LIN {X 21.372,Y -46.394,Z -214.360,A -90.000,B 90.000,C 0.000} C_DIS
LIN {X 21.410,Y -46.395,Z -214.288,A -90.000,B 90.000,C 0.000} C_DIS
LIN {X 22.139,Y -46.405,Z -212.980,A -90.000,B 90.000,C 0.000} C_DIS
LIN {X 23.006,Y -46.442,Z -211.414,A -90.000,B 90.000,C 0.000} C_DIS
LIN {X 23.076,Y -46.443,Z -211.265,A -90.000,B 90.000,C 0.000} C_DIS
LIN {X 23.531,Y -46.448,Z -210.300,A -90.000,B 90.000,C 0.000} C_DIS
LIN {X 23.803,Y -46.447,Z -209.727,A -90.000,B 90.000,C 0.000} C_DIS
LIN {X 23.886,Y -46.448,Z -209.562,A -90.000,B 90.000,C 0.000} C_DIS
LIN {X 24.095,Y -46.453,Z -209.183,A -90.000,B 90.000,C 0.000} C_DIS
LIN {X 24.771,Y -46.497,Z -207.945,A -90.000,B 90.000,C 0.000} C_DIS
LIN {X 25.699,Y -46.521,Z -205.750,A -90.000,B 90.000,C 0.000} C_DIS
LIN {X 25.881,Y -46.530,Z -205.318,A -90.000,B 90.000,C 0.000} C_DIS
LIN {X 25.921,Y -46.533,Z -205.229,A -90.000,B 90.000,C 0.000} C_DIS
LIN {X 26.008,Y -46.539,Z -205.045,A -90.000,B 90.000,C 0.000} C_DIS
LIN {X 26.305,Y -46.563,Z -204.477,A -90.000,B 90.000,C 0.000} C_DIS
LIN {X 27.039,Y -46.567,Z -202.392,A -90.000,B 90.000,C 0.000} C_DIS
LIN {X 27.139,Y -46.575,Z -202.102,A -90.000,B 90.000,C 0.000} C_DIS
LIN {X 27.190,Y -46.580,Z -201.966,A -90.000,B 90.000,C 0.000} C_DIS
LIN {X 27.307,Y -46.591,Z -201.675,A -90.000,B 90.000,C 0.000} C_DIS
LIN {X 27.511,Y -46.604,Z -201.180,A -90.000,B 90.000,C 0.000} C_DIS
LIN {X 27.571,Y -46.605,Z -201.006,A -90.000,B 90.000,C 0.000} C_DIS
LIN {X 28.124,Y -46.633,Z -199.578,A -90.000,B 90.000,C 0.000} C_DIS
LIN {X 28.654,Y -46.698,Z -198.194,A -90.000,B 90.000,C 0.000} C_DIS
LIN {X 28.710,Y -46.701,Z -197.852,A -90.000,B 90.000,C 0.000} C_DIS
LIN {X 28.735,Y -46.703,Z -197.715,A -90.000,B 90.000,C 0.000} C_DIS
LIN {X 28.787,Y -46.703,Z -197.474,A -90.000,B 90.000,C 0.000} C_DIS
LIN {X 28.830,Y -46.702,Z -197.310,A -90.000,B 90.000,C 0.000} C_DIS
LIN {X 28.907,Y -46.704,Z -197.051,A -90.000,B 90.000,C 0.000} C_DIS
LIN {X 28.955,Y -46.705,Z -196.908,A -90.000,B 90.000,C 0.000} C_DIS
LIN {X 28.991,Y -46.707,Z -196.811,A -90.000,B 90.000,C 0.000} C_DIS
LIN {X 29.142,Y -46.723,Z -196.407,A -90.000,B 90.000,C 0.000} C_DIS
LIN {X 29.586,Y -46.772,Z -195.213,A -90.000,B 90.000,C 0.000} C_DIS
LIN {X 29.692,Y -46.777,Z -194.390,A -90.000,B 90.000,C 0.000} C_DIS
LIN {X 29.724,Y -46.775,Z -194.150,A -90.000,B 90.000,C 0.000} C_DIS
LIN {X 29.755,Y -46.774,Z -193.950,A -90.000,B 90.000,C 0.000} C_DIS
LIN {X 29.791,Y -46.774,Z -193.778,A -90.000,B 90.000,C 0.000} C_DIS
LIN {X 29.849,Y -46.771,Z -193.528,A -90.000,B 90.000,C 0.000} C_DIS
LIN {X 29.909,Y -46.770,Z -193.322,A -90.000,B 90.000,C 0.000} C_DIS
LIN {X 30.005,Y -46.772,Z -193.045,A -90.000,B 90.000,C 0.000} C_DIS
LIN {X 30.045,Y -46.774,Z -192.940,A -90.000,B 90.000,C 0.000} C_DIS
LIN {X 30.440,Y -46.794,Z -192.024,A -90.000,B 90.000,C 0.000} C_DIS
LIN {X 30.607,Y -46.786,Z -191.348,A -90.000,B 90.000,C 0.000} C_DIS
LIN {X 30.867,Y -46.781,Z -190.293,A -90.000,B 90.000,C 0.000} C_DIS
LIN {X 30.931,Y -46.768,Z -190.045,A -90.000,B 90.000,C 0.000} C_DIS
LIN {X 30.984,Y -46.760,Z -189.864,A -90.000,B 90.000,C 0.000} C_DIS
LIN {X 31.022,Y -46.755,Z -189.755,A -90.000,B 90.000,C 0.000} C_DIS
LIN {X 31.063,Y -46.752,Z -189.652,A -90.000,B 90.000,C 0.000} C_DIS
LIN {X 31.205,Y -46.744,Z -189.325,A -90.000,B 90.000,C 0.000} C_DIS
LIN {X 31.289,Y -46.742,Z -189.154,A -90.000,B 90.000,C 0.000} C_DIS
LIN {X 31.369,Y -46.741,Z -189.007,A -90.000,B 90.000,C 0.000} C_DIS
LIN {X 31.446,Y -46.742,Z -188.873,A -90.000,B 90.000,C 0.000} C_DIS
LIN {X 32.587,Y -46.759,Z -187.003,A -90.000,B 90.000,C 0.000} C_DIS
LIN {X 32.791,Y -46.747,Z -186.673,A -90.000,B 90.000,C 0.000} C_DIS
LIN {X 33.316,Y -46.732,Z -185.855,A -90.000,B 90.000,C 0.000} C_DIS
LIN {X 33.401,Y -46.731,Z -185.733,A -90.000,B 90.000,C 0.000} C_DIS
LIN {X 33.661,Y -46.733,Z -185.402,A -90.000,B 90.000,C 0.000} C_DIS
LIN {X 33.785,Y -46.734,Z -185.258,A -90.000,B 90.000,C 0.000} C_DIS
LIN {X 34.471,Y -46.751,Z -184.535,A -90.000,B 90.000,C 0.000} C_DIS
LIN {X 34.825,Y -46.750,Z -184.164,A -90.000,B 90.000,C 0.000} C_DIS
LIN {X 35.732,Y -46.716,Z -183.029,A -90.000,B 90.000,C 0.000} C_DIS
LIN {X 35.800,Y -46.714,Z -182.948,A -90.000,B 90.000,C 0.000} C_DIS
LIN {X 35.940,Y -46.711,Z -182.790,A -90.000,B 90.000,C 0.000} C_DIS
LIN {X 36.016,Y -46.709,Z -182.708,A -90.000,B 90.000,C 0.000} C_DIS
LIN {X 36.178,Y -46.712,Z -182.543,A -90.000,B 90.000,C 0.000} C_DIS
LIN {X 36.250,Y -46.714,Z -182.474,A -90.000,B 90.000,C 0.000} C_DIS
LIN {X 36.562,Y -46.723,Z -182.187,A -90.000,B 90.000,C 0.000} C_DIS
LIN {X 37.366,Y -46.703,Z -181.213,A -90.000,B 90.000,C 0.000} C_DIS
LIN {X 37.686,Y -46.706,Z -180.823,A -90.000,B 90.000,C 0.000} C_DIS
LIN {X 37.844,Y -46.709,Z -180.642,A -90.000,B 90.000,C 0.000} C_DIS
LIN {X 38.033,Y -46.714,Z -180.443,A -90.000,B 90.000,C 0.000} C_DIS
LIN {X 38.227,Y -46.722,Z -180.255,A -90.000,B 90.000,C 0.000} C_DIS
LIN {X 38.712,Y -46.742,Z -179.794,A -90.000,B 90.000,C 0.000} C_DIS
LIN {X 39.003,Y -46.762,Z -179.516,A -90.000,B 90.000,C 0.000} C_DIS
LIN {X 39.512,Y -46.791,Z -179.030,A -90.000,B 90.000,C 0.000} C_DIS
LIN {X 39.791,Y -46.799,Z -178.695,A -90.000,B 90.000,C 0.000} C_DIS
LIN {X 39.988,Y -46.805,Z -178.453,A -90.000,B 90.000,C 0.000} C_DIS
LIN {X 40.297,Y -46.807,Z -178.072,A -90.000,B 90.000,C 0.000} C_DIS
LIN {X 40.595,Y -46.815,Z -177.702,A -90.000,B 90.000,C 0.000} C_DIS
LIN {X 41.390,Y -46.827,Z -176.606,A -90.000,B 90.000,C 0.000} C_DIS
LIN {X 41.724,Y -46.832,Z -176.114,A -90.000,B 90.000,C 0.000} C_DIS
LIN {X 42.806,Y -46.849,Z -174.449,A -90.000,B 90.000,C 0.000} C_DIS
LIN {X 42.874,Y -46.850,Z -174.341,A -90.000,B 90.000,C 0.000} C_DIS
LIN {X 43.370,Y -46.859,Z -173.506,A -90.000,B 90.000,C 0.000} C_DIS
LIN {X 44.139,Y -46.868,Z -172.255,A -90.000,B 90.000,C 0.000} C_DIS
LIN {X 44.460,Y -46.875,Z -171.698,A -90.000,B 90.000,C 0.000} C_DIS
LIN {X 44.544,Y -46.876,Z -171.552,A -90.000,B 90.000,C 0.000} C_DIS
LIN {X 44.700,Y -46.881,Z -171.303,A -90.000,B 90.000,C 0.000} C_DIS
LIN {X 44.806,Y -46.885,Z -171.151,A -90.000,B 90.000,C 0.000} C_DIS
LIN {X 44.945,Y -46.893,Z -170.968,A -90.000,B 90.000,C 0.000} C_DIS
LIN {X 45.013,Y -46.896,Z -170.884,A -90.000,B 90.000,C 0.000} C_DIS
LIN {X 45.102,Y -46.902,Z -170.782,A -90.000,B 90.000,C 0.000} C_DIS
LIN {X 45.205,Y -46.909,Z -170.673,A -90.000,B 90.000,C 0.000} C_DIS
LIN {X 45.388,Y -46.923,Z -170.496,A -90.000,B 90.000,C 0.000} C_DIS
LIN {X 45.474,Y -46.930,Z -170.421,A -90.000,B 90.000,C 0.000} C_DIS
LIN {X 45.610,Y -46.942,Z -170.310,A -90.000,B 90.000,C 0.000} C_DIS
LIN {X 45.742,Y -46.955,Z -170.211,A -90.000,B 90.000,C 0.000} C_DIS
LIN {X 45.915,Y -46.972,Z -170.093,A -90.000,B 90.000,C 0.000} C_DIS
LIN {X 47.150,Y -47.044,Z -169.316,A -90.000,B 90.000,C 0.000} C_DIS
LIN {X 48.247,Y -47.104,Z -168.572,A -90.000,B 90.000,C 0.000} C_DIS
LIN {X 48.415,Y -47.114,Z -168.462,A -90.000,B 90.000,C 0.000} C_DIS
LIN {X 48.746,Y -47.121,Z -168.040,A -90.000,B 90.000,C 0.000} C_DIS
LIN {X 48.885,Y -47.126,Z -167.874,A -90.000,B 90.000,C 0.000} C_DIS
LIN {X 48.965,Y -47.129,Z -167.783,A -90.000,B 90.000,C 0.000} C_DIS
LIN {X 49.085,Y -47.134,Z -167.660,A -90.000,B 90.000,C 0.000} C_DIS
LIN {X 49.198,Y -47.140,Z -167.558,A -90.000,B 90.000,C 0.000} C_DIS
LIN {X 49.469,Y -47.154,Z -167.331,A -90.000,B 90.000,C 0.000} C_DIS
LIN {X 49.545,Y -47.158,Z -167.271,A -90.000,B 90.000,C 0.000} C_DIS
LIN {X 49.763,Y -47.167,Z -167.118,A -90.000,B 90.000,C 0.000} C_DIS
LIN {X 49.900,Y -47.173,Z -167.026,A -90.000,B 90.000,C 0.000} C_DIS
LIN {X 50.150,Y -47.184,Z -166.876,A -90.000,B 90.000,C 0.000} C_DIS
LIN {X 50.219,Y -47.186,Z -166.840,A -90.000,B 90.000,C 0.000} C_DIS
LIN {X 50.351,Y -47.187,Z -166.775,A -90.000,B 90.000,C 0.000} C_DIS
LIN {X 50.601,Y -47.189,Z -166.668,A -90.000,B 90.000,C 0.000} C_DIS
LIN {X 50.724,Y -47.190,Z -166.620,A -90.000,B 90.000,C 0.000} C_DIS
LIN {X 50.902,Y -47.192,Z -166.561,A -90.000,B 90.000,C 0.000} C_DIS
LIN {X 51.090,Y -47.195,Z -166.509,A -90.000,B 90.000,C 0.000} C_DIS
LIN {X 51.223,Y -47.197,Z -166.478,A -90.000,B 90.000,C 0.000} C_DIS
LIN {X 51.386,Y -47.202,Z -166.453,A -90.000,B 90.000,C 0.000} C_DIS
LIN {X 51.743,Y -47.213,Z -166.406,A -90.000,B 90.000,C 0.000} C_DIS
LIN {X 51.837,Y -47.216,Z -166.396,A -90.000,B 90.000,C 0.000} C_DIS
LIN {X 51.914,Y -47.218,Z -166.391,A -90.000,B 90.000,C 0.000} C_DIS
LIN {X 52.074,Y -47.224,Z -166.388,A -90.000,B 90.000,C 0.000} C_DIS
LIN {X 52.184,Y -47.228,Z -166.390,A -90.000,B 90.000,C 0.000} C_DIS
LIN {X 52.334,Y -47.233,Z -166.397,A -90.000,B 90.000,C 0.000} C_DIS
LIN {X 52.543,Y -47.241,Z -166.416,A -90.000,B 90.000,C 0.000} C_DIS
LIN {X 52.737,Y -47.248,Z -166.445,A -90.000,B 90.000,C 0.000} C_DIS
LIN {X 52.830,Y -47.251,Z -166.462,A -90.000,B 90.000,C 0.000} C_DIS
LIN {X 53.009,Y -47.258,Z -166.501,A -90.000,B 90.000,C 0.000} C_DIS
LIN {X 53.088,Y -47.261,Z -166.522,A -90.000,B 90.000,C 0.000} C_DIS
LIN {X 53.235,Y -47.264,Z -166.563,A -90.000,B 90.000,C 0.000} C_DIS
LIN {X 53.381,Y -47.262,Z -166.611,A -90.000,B 90.000,C 0.000} C_DIS
LIN {X 53.480,Y -47.257,Z -166.648,A -90.000,B 90.000,C 0.000} C_DIS
LIN {X 53.637,Y -47.250,Z -166.710,A -90.000,B 90.000,C 0.000} C_DIS
LIN {X 53.840,Y -47.240,Z -166.805,A -90.000,B 90.000,C 0.000} C_DIS
LIN {X 53.971,Y -47.234,Z -166.872,A -90.000,B 90.000,C 0.000} C_DIS
LIN {X 54.167,Y -47.224,Z -166.990,A -90.000,B 90.000,C 0.000} C_DIS
LIN {X 54.306,Y -47.219,Z -167.076,A -90.000,B 90.000,C 0.000} C_DIS
LIN {X 54.440,Y -47.213,Z -167.172,A -90.000,B 90.000,C 0.000} C_DIS
LIN {X 54.546,Y -47.209,Z -167.254,A -90.000,B 90.000,C 0.000} C_DIS
LIN {X 54.684,Y -47.203,Z -167.367,A -90.000,B 90.000,C 0.000} C_DIS
LIN {X 54.771,Y -47.199,Z -167.448,A -90.000,B 90.000,C 0.000} C_DIS
LIN {X 54.907,Y -47.194,Z -167.577,A -90.000,B 90.000,C 0.000} C_DIS
LIN {X 55.081,Y -47.186,Z -167.767,A -90.000,B 90.000,C 0.000} C_DIS
LIN {X 55.143,Y -47.183,Z -167.838,A -90.000,B 90.000,C 0.000} C_DIS
LIN {X 55.209,Y -47.180,Z -167.921,A -90.000,B 90.000,C 0.000} C_DIS
LIN {X 55.317,Y -47.175,Z -168.064,A -90.000,B 90.000,C 0.000} C_DIS
LIN {X 55.406,Y -47.171,Z -168.195,A -90.000,B 90.000,C 0.000} C_DIS
LIN {X 55.537,Y -47.165,Z -168.411,A -90.000,B 90.000,C 0.000} C_DIS
LIN {X 55.626,Y -47.160,Z -168.579,A -90.000,B 90.000,C 0.000} C_DIS
LIN {X 55.734,Y -47.155,Z -168.807,A -90.000,B 90.000,C 0.000} C_DIS
LIN {X 55.783,Y -47.149,Z -168.928,A -90.000,B 90.000,C 0.000} C_DIS
LIN {X 55.869,Y -47.136,Z -169.161,A -90.000,B 90.000,C 0.000} C_DIS
LIN {X 55.915,Y -47.130,Z -169.299,A -90.000,B 90.000,C 0.000} C_DIS
LIN {X 55.986,Y -47.119,Z -169.530,A -90.000,B 90.000,C 0.000} C_DIS
LIN {X 56.034,Y -47.109,Z -169.718,A -90.000,B 90.000,C 0.000} C_DIS
LIN {X 56.062,Y -47.102,Z -169.849,A -90.000,B 90.000,C 0.000} C_DIS
LIN {X 56.086,Y -47.093,Z -170.031,A -90.000,B 90.000,C 0.000} C_DIS
LIN {X 56.130,Y -47.074,Z -170.524,A -90.000,B 90.000,C 0.000} C_DIS
LIN {X 56.133,Y -47.064,Z -170.838,A -90.000,B 90.000,C 0.000} C_DIS
LIN {X 56.128,Y -47.063,Z -170.904,A -90.000,B 90.000,C 0.000} C_DIS
LIN {X 56.113,Y -47.059,Z -171.088,A -90.000,B 90.000,C 0.000} C_DIS
LIN {X 55.982,Y -47.036,Z -172.370,A -90.000,B 90.000,C 0.000} C_DIS
LIN {X 55.985,Y -47.029,Z -172.609,A -90.000,B 90.000,C 0.000} C_DIS
LIN {X 55.983,Y -47.020,Z -172.904,A -90.000,B 90.000,C 0.000} C_DIS
LIN {X 55.968,Y -46.990,Z -174.748,A -90.000,B 90.000,C 0.000} C_DIS
LIN {X 56.194,Y -46.944,Z -175.853,A -90.000,B 90.000,C 0.000} C_DIS
LIN {X 56.392,Y -46.920,Z -176.820,A -90.000,B 90.000,C 0.000} C_DIS
LIN {X 56.413,Y -46.917,Z -176.933,A -90.000,B 90.000,C 0.000} C_DIS
LIN {X 56.435,Y -46.914,Z -177.003,A -90.000,B 90.000,C 0.000} C_DIS
LIN {X 56.482,Y -46.909,Z -177.157,A -90.000,B 90.000,C 0.000} C_DIS
LIN {X 56.519,Y -46.904,Z -177.291,A -90.000,B 90.000,C 0.000} C_DIS
LIN {X 56.541,Y -46.902,Z -177.397,A -90.000,B 90.000,C 0.000} C_DIS
LIN {X 56.610,Y -46.893,Z -177.772,A -90.000,B 90.000,C 0.000} C_DIS
LIN {X 56.630,Y -46.890,Z -177.901,A -90.000,B 90.000,C 0.000} C_DIS
LIN {X 56.698,Y -46.865,Z -178.691,A -90.000,B 90.000,C 0.000} C_DIS
LIN {X 56.729,Y -46.861,Z -179.054,A -90.000,B 90.000,C 0.000} C_DIS
LIN {X 56.742,Y -46.858,Z -179.247,A -90.000,B 90.000,C 0.000} C_DIS
LIN {X 56.766,Y -46.850,Z -180.111,A -90.000,B 90.000,C 0.000} C_DIS
LIN {X 56.805,Y -46.843,Z -180.308,A -90.000,B 90.000,C 0.000} C_DIS
LIN {X 56.834,Y -46.838,Z -180.478,A -90.000,B 90.000,C 0.000} C_DIS
LIN {X 56.860,Y -46.833,Z -180.668,A -90.000,B 90.000,C 0.000} C_DIS
LIN {X 56.942,Y -46.816,Z -181.375,A -90.000,B 90.000,C 0.000} C_DIS
LIN {X 57.059,Y -46.811,Z -182.378,A -90.000,B 90.000,C 0.000} C_DIS
LIN {X 57.260,Y -46.789,Z -183.172,A -90.000,B 90.000,C 0.000} C_DIS
LIN {X 57.464,Y -46.761,Z -183.982,A -90.000,B 90.000,C 0.000} C_DIS
LIN {X 57.683,Y -46.740,Z -184.857,A -90.000,B 90.000,C 0.000} C_DIS
LIN {X 57.706,Y -46.738,Z -184.961,A -90.000,B 90.000,C 0.000} C_DIS
LIN {X 57.750,Y -46.735,Z -185.198,A -90.000,B 90.000,C 0.000} C_DIS
LIN {X 57.780,Y -46.730,Z -185.418,A -90.000,B 90.000,C 0.000} C_DIS
LIN {X 57.792,Y -46.728,Z -185.529,A -90.000,B 90.000,C 0.000} C_DIS
LIN {X 57.810,Y -46.725,Z -185.751,A -90.000,B 90.000,C 0.000} C_DIS
LIN {X 57.816,Y -46.724,Z -185.862,A -90.000,B 90.000,C 0.000} C_DIS
LIN {X 57.830,Y -46.723,Z -186.394,A -90.000,B 90.000,C 0.000} C_DIS
LIN {X 57.878,Y -46.697,Z -188.394,A -90.000,B 90.000,C 0.000} C_DIS
LIN {X 57.892,Y -46.688,Z -189.117,A -90.000,B 90.000,C 0.000} C_DIS
LIN {X 57.901,Y -46.676,Z -189.755,A -90.000,B 90.000,C 0.000} C_DIS
LIN {X 57.886,Y -46.667,Z -190.472,A -90.000,B 90.000,C 0.000} C_DIS
LIN {X 57.861,Y -46.650,Z -191.585,A -90.000,B 90.000,C 0.000} C_DIS
LIN {X 57.817,Y -46.643,Z -192.376,A -90.000,B 90.000,C 0.000} C_DIS
LIN {X 57.692,Y -46.603,Z -194.422,A -90.000,B 90.000,C 0.000} C_DIS
LIN {X 57.613,Y -46.589,Z -195.317,A -90.000,B 90.000,C 0.000} C_DIS
LIN {X 57.579,Y -46.587,Z -195.575,A -90.000,B 90.000,C 0.000} C_DIS
LIN {X 57.518,Y -46.584,Z -195.936,A -90.000,B 90.000,C 0.000} C_DIS
LIN {X 57.317,Y -46.558,Z -197.358,A -90.000,B 90.000,C 0.000} C_DIS
LIN {X 57.301,Y -46.557,Z -197.457,A -90.000,B 90.000,C 0.000} C_DIS
LIN {X 57.263,Y -46.555,Z -197.652,A -90.000,B 90.000,C 0.000} C_DIS
LIN {X 57.242,Y -46.555,Z -197.750,A -90.000,B 90.000,C 0.000} C_DIS
LIN {X 56.835,Y -46.557,Z -199.423,A -90.000,B 90.000,C 0.000} C_DIS
LIN {X 56.752,Y -46.556,Z -199.758,A -90.000,B 90.000,C 0.000} C_DIS
LIN {X 56.657,Y -46.556,Z -200.089,A -90.000,B 90.000,C 0.000} C_DIS
LIN {X 55.436,Y -46.517,Z -204.266,A -90.000,B 90.000,C 0.000} C_DIS
LIN {X 55.255,Y -46.511,Z -204.846,A -90.000,B 90.000,C 0.000} C_DIS
LIN {X 53.989,Y -46.479,Z -208.784,A -90.000,B 90.000,C 0.000} C_DIS
LIN {X 53.153,Y -46.455,Z -211.322,A -90.000,B 90.000,C 0.000} C_DIS
LIN {X 52.318,Y -46.436,Z -213.780,A -90.000,B 90.000,C 0.000} C_DIS
LIN {X 51.568,Y -46.421,Z -215.923,A -90.000,B 90.000,C 0.000} C_DIS
LIN {X 50.680,Y -46.391,Z -218.613,A -90.000,B 90.000,C 0.000} C_DIS
LIN {X 50.512,Y -46.383,Z -219.120,A -90.000,B 90.000,C 0.000} C_DIS
LIN {X 50.421,Y -46.380,Z -219.365,A -90.000,B 90.000,C 0.000} C_DIS
LIN {X 49.901,Y -46.375,Z -220.611,A -90.000,B 90.000,C 0.000} C_DIS
LIN {X 48.449,Y -46.347,Z -224.309,A -90.000,B 90.000,C 0.000} C_DIS
LIN {X 48.296,Y -46.336,Z -224.688,A -90.000,B 90.000,C 0.000} C_DIS
LIN {X 48.260,Y -46.334,Z -224.769,A -90.000,B 90.000,C 0.000} C_DIS
LIN {X 48.153,Y -46.332,Z -224.986,A -90.000,B 90.000,C 0.000} C_DIS
LIN {X 47.797,Y -46.334,Z -225.635,A -90.000,B 90.000,C 0.000} C_DIS
LIN {X 45.651,Y -46.342,Z -229.733,A -90.000,B 90.000,C 0.000} C_DIS
LIN {X 45.386,Y -46.325,Z -230.225,A -90.000,B 90.000,C 0.000} C_DIS
LIN {X 45.319,Y -46.322,Z -230.340,A -90.000,B 90.000,C 0.000} C_DIS
LIN {X 45.240,Y -46.320,Z -230.470,A -90.000,B 90.000,C 0.000} C_DIS
LIN {X 45.141,Y -46.319,Z -230.620,A -90.000,B 90.000,C 0.000} C_DIS
LIN {X 45.007,Y -46.319,Z -230.811,A -90.000,B 90.000,C 0.000} C_DIS
LIN {X 44.913,Y -46.321,Z -230.936,A -90.000,B 90.000,C 0.000} C_DIS
LIN {X 44.469,Y -46.335,Z -231.506,A -90.000,B 90.000,C 0.000} C_DIS
LIN {X 42.222,Y -46.392,Z -234.502,A -90.000,B 90.000,C 0.000} C_DIS
LIN {X 42.075,Y -46.396,Z -234.697,A -90.000,B 90.000,C 0.000} C_DIS
LIN {X 41.938,Y -46.393,Z -234.877,A -90.000,B 90.000,C 0.000} C_DIS
LIN {X 41.279,Y -46.363,Z -235.736,A -90.000,B 90.000,C 0.000} C_DIS
LIN {X 41.178,Y -46.359,Z -235.859,A -90.000,B 90.000,C 0.000} C_DIS
LIN {X 40.922,Y -46.359,Z -236.132,A -90.000,B 90.000,C 0.000} C_DIS
LIN {X 40.816,Y -46.361,Z -236.236,A -90.000,B 90.000,C 0.000} C_DIS
LIN {X 40.535,Y -46.369,Z -236.493,A -90.000,B 90.000,C 0.000} C_DIS
LIN {X 39.541,Y -46.410,Z -237.341,A -90.000,B 90.000,C 0.000} C_DIS
LIN {X 37.363,Y -46.508,Z -239.204,A -90.000,B 90.000,C 0.000} C_DIS
LIN {X 37.190,Y -46.515,Z -239.357,A -90.000,B 90.000,C 0.000} C_DIS
LIN {X 35.620,Y -46.514,Z -240.714,A -90.000,B 90.000,C 0.000} C_DIS
LIN {X 35.453,Y -46.516,Z -240.850,A -90.000,B 90.000,C 0.000} C_DIS
LIN {X 35.099,Y -46.524,Z -241.116,A -90.000,B 90.000,C 0.000} C_DIS
LIN {X 34.884,Y -46.532,Z -241.266,A -90.000,B 90.000,C 0.000} C_DIS
LIN {X 34.639,Y -46.540,Z -241.425,A -90.000,B 90.000,C 0.000} C_DIS
LIN {X 34.019,Y -46.542,Z -241.822,A -90.000,B 90.000,C 0.000} C_DIS
LIN {X 32.974,Y -46.548,Z -242.464,A -90.000,B 90.000,C 0.000} C_DIS
LIN {X 32.749,Y -46.551,Z -242.591,A -90.000,B 90.000,C 0.000} C_DIS
LIN {X 32.635,Y -46.554,Z -242.650,A -90.000,B 90.000,C 0.000} C_DIS
LIN {X 32.446,Y -46.559,Z -242.740,A -90.000,B 90.000,C 0.000} C_DIS
LIN {X 32.356,Y -46.562,Z -242.780,A -90.000,B 90.000,C 0.000} C_DIS
LIN {X 32.151,Y -46.569,Z -242.866,A -90.000,B 90.000,C 0.000} C_DIS
LIN {X 32.047,Y -46.574,Z -242.906,A -90.000,B 90.000,C 0.000} C_DIS
LIN {X 30.994,Y -46.623,Z -243.279,A -90.000,B 90.000,C 0.000} C_DIS
LIN {X 30.191,Y -46.651,Z -243.561,A -90.000,B 90.000,C 0.000} C_DIS
LIN {X 30.191,Y -60.000,Z -243.561,A -90.000,B 90.000,C 0.000} C_DIS
LIN {X 14.010,Y -60.000,Z -243.561,A -90.000,B 90.000,C 0.000} C_DIS
LIN {X 14.010,Y -46.891,Z -243.561,A -90.000,B 90.000,C 0.000} C_DIS
LIN {X 13.959,Y -46.892,Z -243.476,A -90.000,B 90.000,C 0.000} C_DIS
LIN {X 13.510,Y -46.904,Z -242.722,A -90.000,B 90.000,C 0.000} C_DIS
LIN {X 13.086,Y -46.925,Z -242.012,A -90.000,B 90.000,C 0.000} C_DIS
LIN {X 13.052,Y -46.925,Z -241.955,A -90.000,B 90.000,C 0.000} C_DIS
LIN {X 12.810,Y -46.904,Z -241.545,A -90.000,B 90.000,C 0.000} C_DIS
LIN {X 11.960,Y -46.805,Z -240.098,A -90.000,B 90.000,C 0.000} C_DIS
LIN {X 11.830,Y -46.789,Z -239.865,A -90.000,B 90.000,C 0.000} C_DIS
LIN {X 11.709,Y -46.775,Z -239.631,A -90.000,B 90.000,C 0.000} C_DIS
LIN {X 11.634,Y -46.765,Z -239.474,A -90.000,B 90.000,C 0.000} C_DIS
LIN {X 11.525,Y -46.751,Z -239.218,A -90.000,B 90.000,C 0.000} C_DIS
LIN {X 11.453,Y -46.742,Z -239.014,A -90.000,B 90.000,C 0.000} C_DIS
LIN {X 11.292,Y -46.719,Z -238.497,A -90.000,B 90.000,C 0.000} C_DIS
LIN {X 11.251,Y -46.712,Z -238.354,A -90.000,B 90.000,C 0.000} C_DIS
LIN {X 11.212,Y -46.706,Z -238.196,A -90.000,B 90.000,C 0.000} C_DIS
LIN {X 11.178,Y -46.700,Z -238.026,A -90.000,B 90.000,C 0.000} C_DIS
LIN {X 11.155,Y -46.696,Z -237.892,A -90.000,B 90.000,C 0.000} C_DIS
LIN {X 11.094,Y -46.683,Z -237.451,A -90.000,B 90.000,C 0.000} C_DIS
LIN {X 11.069,Y -46.663,Z -237.257,A -90.000,B 90.000,C 0.000} C_DIS
LIN {X 11.043,Y -46.634,Z -236.968,A -90.000,B 90.000,C 0.000} C_DIS
LIN {X 11.032,Y -46.619,Z -236.802,A -90.000,B 90.000,C 0.000} C_DIS
LIN {X 11.022,Y -46.594,Z -236.521,A -90.000,B 90.000,C 0.000} C_DIS
LIN {X 11.021,Y -46.584,Z -236.407,A -90.000,B 90.000,C 0.000} C_DIS
LIN {X 11.023,Y -46.567,Z -236.192,A -90.000,B 90.000,C 0.000} C_DIS
LIN {X 11.031,Y -46.551,Z -235.982,A -90.000,B 90.000,C 0.000} C_DIS
LIN {X 11.050,Y -46.535,Z -235.754,A -90.000,B 90.000,C 0.000} C_DIS
LIN {X 11.080,Y -46.520,Z -235.513,A -90.000,B 90.000,C 0.000} C_DIS
LIN {X 11.121,Y -46.507,Z -235.265,A -90.000,B 90.000,C 0.000} C_DIS
LIN {X 11.275,Y -46.470,Z -234.509,A -90.000,B 90.000,C 0.000} C_DIS
LIN {X 12.144,Y -46.244,Z -230.270,A -90.000,B 90.000,C 0.000} C_DIS
LIN {X 12.227,Y -46.227,Z -229.912,A -90.000,B 90.000,C 0.000} C_DIS
LIN {X 12.250,Y -46.223,Z -229.820,A -90.000,B 90.000,C 0.000} C_DIS
LIN {X 12.317,Y -46.213,Z -229.582,A -90.000,B 90.000,C 0.000} C_DIS
LIN {X 12.403,Y -46.202,Z -229.309,A -90.000,B 90.000,C 0.000} C_DIS
LIN {X 12.816,Y -46.127,Z -228.037,A -90.000,B 90.000,C 0.000} C_DIS
LIN {X 13.503,Y -46.012,Z -225.913,A -90.000,B 90.000,C 0.000} C_DIS
LIN {X 13.817,Y -45.960,Z -224.949,A -90.000,B 90.000,C 0.000} C_DIS
LIN {X 13.883,Y -45.951,Z -224.768,A -90.000,B 90.000,C 0.000} C_DIS
LIN {X 13.944,Y -45.945,Z -224.611,A -90.000,B 90.000,C 0.000} C_DIS
LIN {X 14.233,Y -45.925,Z -223.939,A -90.000,B 90.000,C 0.000} C_DIS
LIN {X 14.390,Y -45.916,Z -223.580,A -90.000,B 90.000,C 0.000} C_DIS
LIN {X 15.194,Y -45.890,Z -221.928,A -90.000,B 90.000,C 0.000} C_DIS
LIN {X 16.760,Y -45.862,Z -218.903,A -90.000,B 90.000,C 0.000} C_DIS
LIN {X 17.047,Y -45.860,Z -218.348,A -90.000,B 90.000,C 0.000} C_DIS
LIN {X 17.879,Y -45.873,Z -216.819,A -90.000,B 90.000,C 0.000} C_DIS
LIN {X 19.013,Y -45.885,Z -214.742,A -90.000,B 90.000,C 0.000} C_DIS
LIN {X 19.214,Y -45.885,Z -214.344,A -90.000,B 90.000,C 0.000} C_DIS
LIN {X 19.645,Y -45.890,Z -213.488,A -90.000,B 90.000,C 0.000} C_DIS
LIN {X 19.683,Y -45.891,Z -213.415,A -90.000,B 90.000,C 0.000} C_DIS
LIN {X 20.993,Y -45.936,Z -211.047,A -90.000,B 90.000,C 0.000} C_DIS
LIN {X 21.281,Y -45.952,Z -210.524,A -90.000,B 90.000,C 0.000} C_DIS
LIN {X 22.048,Y -45.971,Z -208.895,A -90.000,B 90.000,C 0.000} C_DIS
LIN {X 22.185,Y -45.977,Z -208.623,A -90.000,B 90.000,C 0.000} C_DIS
LIN {X 22.868,Y -46.015,Z -207.373,A -90.000,B 90.000,C 0.000} C_DIS
LIN {X 23.022,Y -46.028,Z -207.089,A -90.000,B 90.000,C 0.000} C_DIS
LIN {X 23.669,Y -46.062,Z -205.549,A -90.000,B 90.000,C 0.000} C_DIS
LIN {X 24.057,Y -46.079,Z -204.630,A -90.000,B 90.000,C 0.000} C_DIS
LIN {X 24.145,Y -46.083,Z -204.427,A -90.000,B 90.000,C 0.000} C_DIS
LIN {X 24.253,Y -46.090,Z -204.197,A -90.000,B 90.000,C 0.000} C_DIS
LIN {X 24.514,Y -46.120,Z -203.690,A -90.000,B 90.000,C 0.000} C_DIS
LIN {X 25.133,Y -46.172,Z -201.901,A -90.000,B 90.000,C 0.000} C_DIS
LIN {X 25.318,Y -46.187,Z -201.374,A -90.000,B 90.000,C 0.000} C_DIS
LIN {X 25.381,Y -46.193,Z -201.207,A -90.000,B 90.000,C 0.000} C_DIS
LIN {X 25.675,Y -46.226,Z -200.481,A -90.000,B 90.000,C 0.000} C_DIS
LIN {X 25.725,Y -46.230,Z -200.334,A -90.000,B 90.000,C 0.000} C_DIS
LIN {X 26.642,Y -46.319,Z -197.945,A -90.000,B 90.000,C 0.000} C_DIS
LIN {X 26.748,Y -46.334,Z -197.667,A -90.000,B 90.000,C 0.000} C_DIS
LIN {X 26.800,Y -46.337,Z -197.364,A -90.000,B 90.000,C 0.000} C_DIS
LIN {X 26.829,Y -46.340,Z -197.222,A -90.000,B 90.000,C 0.000} C_DIS
LIN {X 26.865,Y -46.340,Z -197.058,A -90.000,B 90.000,C 0.000} C_DIS
LIN {X 26.927,Y -46.342,Z -196.812,A -90.000,B 90.000,C 0.000} C_DIS
LIN {X 27.020,Y -46.346,Z -196.493,A -90.000,B 90.000,C 0.000} C_DIS
LIN {X 27.091,Y -46.351,Z -196.276,A -90.000,B 90.000,C 0.000} C_DIS
LIN {X 27.484,Y -46.384,Z -195.219,A -90.000,B 90.000,C 0.000} C_DIS
LIN {X 27.666,Y -46.406,Z -194.730,A -90.000,B 90.000,C 0.000} C_DIS
LIN {X 27.775,Y -46.406,Z -193.896,A -90.000,B 90.000,C 0.000} C_DIS
LIN {X 27.813,Y -46.407,Z -193.646,A -90.000,B 90.000,C 0.000} C_DIS
LIN {X 27.837,Y -46.408,Z -193.520,A -90.000,B 90.000,C 0.000} C_DIS
LIN {X 27.865,Y -46.408,Z -193.381,A -90.000,B 90.000,C 0.000} C_DIS
LIN {X 27.932,Y -46.405,Z -193.089,A -90.000,B 90.000,C 0.000} C_DIS
LIN {X 27.966,Y -46.404,Z -192.962,A -90.000,B 90.000,C 0.000} C_DIS
LIN {X 28.043,Y -46.405,Z -192.699,A -90.000,B 90.000,C 0.000} C_DIS
LIN {X 28.123,Y -46.408,Z -192.468,A -90.000,B 90.000,C 0.000} C_DIS
LIN {X 28.177,Y -46.411,Z -192.317,A -90.000,B 90.000,C 0.000} C_DIS
LIN {X 28.241,Y -46.414,Z -192.155,A -90.000,B 90.000,C 0.000} C_DIS
LIN {X 28.569,Y -46.435,Z -191.392,A -90.000,B 90.000,C 0.000} C_DIS
LIN {X 28.971,Y -46.423,Z -189.765,A -90.000,B 90.000,C 0.000} C_DIS
LIN {X 29.039,Y -46.410,Z -189.503,A -90.000,B 90.000,C 0.000} C_DIS
LIN {X 29.118,Y -46.395,Z -189.244,A -90.000,B 90.000,C 0.000} C_DIS
LIN {X 29.172,Y -46.387,Z -189.089,A -90.000,B 90.000,C 0.000} C_DIS
LIN {X 29.236,Y -46.381,Z -188.927,A -90.000,B 90.000,C 0.000} C_DIS
LIN {X 29.400,Y -46.369,Z -188.549,A -90.000,B 90.000,C 0.000} C_DIS
LIN {X 29.451,Y -46.367,Z -188.442,A -90.000,B 90.000,C 0.000} C_DIS
LIN {X 29.525,Y -46.364,Z -188.291,A -90.000,B 90.000,C 0.000} C_DIS
LIN {X 29.643,Y -46.362,Z -188.071,A -90.000,B 90.000,C 0.000} C_DIS
LIN {X 29.741,Y -46.362,Z -187.899,A -90.000,B 90.000,C 0.000} C_DIS
LIN {X 30.341,Y -46.372,Z -186.913,A -90.000,B 90.000,C 0.000} C_DIS
LIN {X 30.578,Y -46.375,Z -186.525,A -90.000,B 90.000,C 0.000} C_DIS
LIN {X 31.119,Y -46.343,Z -185.653,A -90.000,B 90.000,C 0.000} C_DIS
LIN {X 31.667,Y -46.315,Z -184.804,A -90.000,B 90.000,C 0.000} C_DIS
LIN {X 31.795,Y -46.310,Z -184.619,A -90.000,B 90.000,C 0.000} C_DIS
LIN {X 31.863,Y -46.308,Z -184.528,A -90.000,B 90.000,C 0.000} C_DIS
LIN {X 32.123,Y -46.305,Z -184.197,A -90.000,B 90.000,C 0.000} C_DIS
LIN {X 32.253,Y -46.307,Z -184.041,A -90.000,B 90.000,C 0.000} C_DIS
LIN {X 32.372,Y -46.311,Z -183.907,A -90.000,B 90.000,C 0.000} C_DIS
LIN {X 32.528,Y -46.313,Z -183.743,A -90.000,B 90.000,C 0.000} C_DIS
LIN {X 33.351,Y -46.309,Z -182.883,A -90.000,B 90.000,C 0.000} C_DIS
LIN {X 33.735,Y -46.294,Z -182.402,A -90.000,B 90.000,C 0.000} C_DIS
LIN {X 34.117,Y -46.290,Z -181.920,A -90.000,B 90.000,C 0.000} C_DIS
LIN {X 34.265,Y -46.289,Z -181.736,A -90.000,B 90.000,C 0.000} C_DIS
LIN {X 34.430,Y -46.291,Z -181.546,A -90.000,B 90.000,C 0.000} C_DIS
LIN {X 34.580,Y -46.292,Z -181.380,A -90.000,B 90.000,C 0.000} C_DIS
LIN {X 34.788,Y -46.293,Z -181.168,A -90.000,B 90.000,C 0.000} C_DIS
LIN {X 34.895,Y -46.294,Z -181.064,A -90.000,B 90.000,C 0.000} C_DIS
LIN {X 35.140,Y -46.300,Z -180.838,A -90.000,B 90.000,C 0.000} C_DIS
LIN {X 36.172,Y -46.306,Z -179.579,A -90.000,B 90.000,C 0.000} C_DIS
LIN {X 36.414,Y -46.311,Z -179.302,A -90.000,B 90.000,C 0.000} C_DIS
LIN {X 36.617,Y -46.323,Z -179.087,A -90.000,B 90.000,C 0.000} C_DIS
LIN {X 36.866,Y -46.333,Z -178.842,A -90.000,B 90.000,C 0.000} C_DIS
LIN {X 37.868,Y -46.376,Z -177.890,A -90.000,B 90.000,C 0.000} C_DIS
LIN {X 38.086,Y -46.391,Z -177.682,A -90.000,B 90.000,C 0.000} C_DIS
LIN {X 38.384,Y -46.402,Z -177.320,A -90.000,B 90.000,C 0.000} C_DIS
LIN {X 39.039,Y -46.425,Z -176.506,A -90.000,B 90.000,C 0.000} C_DIS
LIN {X 39.214,Y -46.429,Z -176.265,A -90.000,B 90.000,C 0.000} C_DIS
LIN {X 39.799,Y -46.453,Z -175.453,A -90.000,B 90.000,C 0.000} C_DIS
LIN {X 40.077,Y -46.461,Z -175.041,A -90.000,B 90.000,C 0.000} C_DIS
LIN {X 40.413,Y -46.468,Z -174.525,A -90.000,B 90.000,C 0.000} C_DIS
LIN {X 41.196,Y -46.498,Z -173.312,A -90.000,B 90.000,C 0.000} C_DIS
LIN {X 41.678,Y -46.507,Z -172.498,A -90.000,B 90.000,C 0.000} C_DIS
LIN {X 42.427,Y -46.535,Z -171.273,A -90.000,B 90.000,C 0.000} C_DIS
LIN {X 42.837,Y -46.539,Z -170.565,A -90.000,B 90.000,C 0.000} C_DIS
LIN {X 43.040,Y -46.543,Z -170.240,A -90.000,B 90.000,C 0.000} C_DIS
LIN {X 43.189,Y -46.547,Z -170.022,A -90.000,B 90.000,C 0.000} C_DIS
LIN {X 43.327,Y -46.553,Z -169.838,A -90.000,B 90.000,C 0.000} C_DIS
LIN {X 43.490,Y -46.560,Z -169.632,A -90.000,B 90.000,C 0.000} C_DIS
LIN {X 43.629,Y -46.568,Z -169.471,A -90.000,B 90.000,C 0.000} C_DIS
LIN {X 43.784,Y -46.578,Z -169.305,A -90.000,B 90.000,C 0.000} C_DIS
LIN {X 43.997,Y -46.593,Z -169.097,A -90.000,B 90.000,C 0.000} C_DIS
LIN {X 44.116,Y -46.602,Z -168.986,A -90.000,B 90.000,C 0.000} C_DIS
LIN {X 44.203,Y -46.609,Z -168.911,A -90.000,B 90.000,C 0.000} C_DIS
LIN {X 44.377,Y -46.625,Z -168.767,A -90.000,B 90.000,C 0.000} C_DIS
LIN {X 44.508,Y -46.637,Z -168.667,A -90.000,B 90.000,C 0.000} C_DIS
LIN {X 44.648,Y -46.650,Z -168.565,A -90.000,B 90.000,C 0.000} C_DIS
LIN {X 44.821,Y -46.667,Z -168.447,A -90.000,B 90.000,C 0.000} C_DIS
LIN {X 46.074,Y -46.798,Z -167.648,A -90.000,B 90.000,C 0.000} C_DIS
LIN {X 46.925,Y -46.887,Z -167.065,A -90.000,B 90.000,C 0.000} C_DIS
LIN {X 47.053,Y -46.897,Z -166.978,A -90.000,B 90.000,C 0.000} C_DIS
LIN {X 47.167,Y -46.899,Z -166.833,A -90.000,B 90.000,C 0.000} C_DIS
LIN {X 47.366,Y -46.904,Z -166.591,A -90.000,B 90.000,C 0.000} C_DIS
LIN {X 47.490,Y -46.908,Z -166.452,A -90.000,B 90.000,C 0.000} C_DIS
LIN {X 47.683,Y -46.916,Z -166.250,A -90.000,B 90.000,C 0.000} C_DIS
LIN {X 47.871,Y -46.924,Z -166.077,A -90.000,B 90.000,C 0.000} C_DIS
LIN {X 48.151,Y -46.939,Z -165.841,A -90.000,B 90.000,C 0.000} C_DIS
LIN {X 48.342,Y -46.949,Z -165.687,A -90.000,B 90.000,C 0.000} C_DIS
LIN {X 48.556,Y -46.961,Z -165.534,A -90.000,B 90.000,C 0.000} C_DIS
LIN {X 48.794,Y -46.976,Z -165.371,A -90.000,B 90.000,C 0.000} C_DIS
LIN {X 48.885,Y -46.982,Z -165.313,A -90.000,B 90.000,C 0.000} C_DIS
LIN {X 49.136,Y -46.999,Z -165.162,A -90.000,B 90.000,C 0.000} C_DIS
LIN {X 49.247,Y -47.007,Z -165.100,A -90.000,B 90.000,C 0.000} C_DIS
LIN {X 49.474,Y -47.023,Z -164.985,A -90.000,B 90.000,C 0.000} C_DIS
LIN {X 49.814,Y -47.050,Z -164.834,A -90.000,B 90.000,C 0.000} C_DIS
LIN {X 49.993,Y -47.065,Z -164.762,A -90.000,B 90.000,C 0.000} C_DIS
LIN {X 50.091,Y -47.073,Z -164.726,A -90.000,B 90.000,C 0.000} C_DIS
LIN {X 50.277,Y -47.089,Z -164.664,A -90.000,B 90.000,C 0.000} C_DIS
LIN {X 50.378,Y -47.098,Z -164.633,A -90.000,B 90.000,C 0.000} C_DIS
LIN {X 50.561,Y -47.108,Z -164.582,A -90.000,B 90.000,C 0.000} C_DIS
LIN {X 50.773,Y -47.120,Z -164.531,A -90.000,B 90.000,C 0.000} C_DIS
LIN {X 50.921,Y -47.128,Z -164.503,A -90.000,B 90.000,C 0.000} C_DIS
LIN {X 51.099,Y -47.133,Z -164.475,A -90.000,B 90.000,C 0.000} C_DIS
LIN {X 51.336,Y -47.139,Z -164.444,A -90.000,B 90.000,C 0.000} C_DIS
LIN {X 51.630,Y -47.147,Z -164.408,A -90.000,B 90.000,C 0.000} C_DIS
LIN {X 51.797,Y -47.151,Z -164.395,A -90.000,B 90.000,C 0.000} C_DIS
LIN {X 52.053,Y -47.159,Z -164.389,A -90.000,B 90.000,C 0.000} C_DIS
LIN {X 52.224,Y -47.165,Z -164.391,A -90.000,B 90.000,C 0.000} C_DIS
LIN {X 52.429,Y -47.171,Z -164.400,A -90.000,B 90.000,C 0.000} C_DIS
LIN {X 52.544,Y -47.175,Z -164.409,A -90.000,B 90.000,C 0.000} C_DIS
LIN {X 52.799,Y -47.184,Z -164.434,A -90.000,B 90.000,C 0.000} C_DIS
LIN {X 52.955,Y -47.192,Z -164.456,A -90.000,B 90.000,C 0.000} C_DIS
LIN {X 53.117,Y -47.200,Z -164.482,A -90.000,B 90.000,C 0.000} C_DIS
LIN {X 53.266,Y -47.208,Z -164.510,A -90.000,B 90.000,C 0.000} C_DIS
LIN {X 53.445,Y -47.218,Z -164.550,A -90.000,B 90.000,C 0.000} C_DIS
LIN {X 53.695,Y -47.231,Z -164.615,A -90.000,B 90.000,C 0.000} C_DIS
LIN {X 53.860,Y -47.232,Z -164.663,A -90.000,B 90.000,C 0.000} C_DIS
LIN {X 53.922,Y -47.232,Z -164.684,A -90.000,B 90.000,C 0.000} C_DIS
LIN {X 54.097,Y -47.226,Z -164.743,A -90.000,B 90.000,C 0.000} C_DIS
LIN {X 54.245,Y -47.221,Z -164.800,A -90.000,B 90.000,C 0.000} C_DIS
LIN {X 54.446,Y -47.214,Z -164.882,A -90.000,B 90.000,C 0.000} C_DIS
LIN {X 54.674,Y -47.206,Z -164.987,A -90.000,B 90.000,C 0.000} C_DIS
LIN {X 54.884,Y -47.199,Z -165.093,A -90.000,B 90.000,C 0.000} C_DIS
LIN {X 54.991,Y -47.195,Z -165.153,A -90.000,B 90.000,C 0.000} C_DIS
LIN {X 55.190,Y -47.188,Z -165.271,A -90.000,B 90.000,C 0.000} C_DIS
LIN {X 55.367,Y -47.182,Z -165.381,A -90.000,B 90.000,C 0.000} C_DIS
LIN {X 55.486,Y -47.178,Z -165.462,A -90.000,B 90.000,C 0.000} C_DIS
LIN {X 55.599,Y -47.175,Z -165.542,A -90.000,B 90.000,C 0.000} C_DIS
LIN {X 55.768,Y -47.169,Z -165.671,A -90.000,B 90.000,C 0.000} C_DIS
LIN {X 55.955,Y -47.163,Z -165.823,A -90.000,B 90.000,C 0.000} C_DIS
LIN {X 56.049,Y -47.160,Z -165.907,A -90.000,B 90.000,C 0.000} C_DIS
LIN {X 56.279,Y -47.153,Z -166.122,A -90.000,B 90.000,C 0.000} C_DIS
LIN {X 56.381,Y -47.150,Z -166.226,A -90.000,B 90.000,C 0.000} C_DIS
LIN {X 56.488,Y -47.147,Z -166.342,A -90.000,B 90.000,C 0.000} C_DIS
LIN {X 56.562,Y -47.140,Z -166.423,A -90.000,B 90.000,C 0.000} C_DIS
LIN {X 56.700,Y -47.125,Z -166.584,A -90.000,B 90.000,C 0.000} C_DIS
LIN {X 56.823,Y -47.111,Z -166.743,A -90.000,B 90.000,C 0.000} C_DIS
LIN {X 56.907,Y -47.100,Z -166.853,A -90.000,B 90.000,C 0.000} C_DIS
LIN {X 57.072,Y -47.075,Z -167.092,A -90.000,B 90.000,C 0.000} C_DIS
LIN {X 57.244,Y -47.048,Z -167.375,A -90.000,B 90.000,C 0.000} C_DIS
LIN {X 57.297,Y -47.039,Z -167.470,A -90.000,B 90.000,C 0.000} C_DIS
LIN {X 57.380,Y -47.026,Z -167.627,A -90.000,B 90.000,C 0.000} C_DIS
LIN {X 57.429,Y -47.017,Z -167.725,A -90.000,B 90.000,C 0.000} C_DIS
LIN {X 57.506,Y -47.004,Z -167.888,A -90.000,B 90.000,C 0.000} C_DIS
LIN {X 57.569,Y -46.993,Z -168.028,A -90.000,B 90.000,C 0.000} C_DIS
LIN {X 57.625,Y -46.983,Z -168.166,A -90.000,B 90.000,C 0.000} C_DIS
LIN {X 57.737,Y -46.962,Z -168.469,A -90.000,B 90.000,C 0.000} C_DIS
LIN {X 57.800,Y -46.949,Z -168.654,A -90.000,B 90.000,C 0.000} C_DIS
LIN {X 57.888,Y -46.931,Z -168.942,A -90.000,B 90.000,C 0.000} C_DIS
LIN {X 57.960,Y -46.915,Z -169.216,A -90.000,B 90.000,C 0.000} C_DIS
LIN {X 58.005,Y -46.904,Z -169.418,A -90.000,B 90.000,C 0.000} C_DIS
LIN {X 58.032,Y -46.897,Z -169.575,A -90.000,B 90.000,C 0.000} C_DIS
LIN {X 58.057,Y -46.888,Z -169.757,A -90.000,B 90.000,C 0.000} C_DIS
LIN {X 58.075,Y -46.881,Z -169.944,A -90.000,B 90.000,C 0.000} C_DIS
LIN {X 58.111,Y -46.864,Z -170.350,A -90.000,B 90.000,C 0.000} C_DIS
LIN {X 58.117,Y -46.861,Z -170.441,A -90.000,B 90.000,C 0.000} C_DIS
LIN {X 58.121,Y -46.847,Z -170.836,A -90.000,B 90.000,C 0.000} C_DIS
LIN {X 58.116,Y -46.843,Z -170.970,A -90.000,B 90.000,C 0.000} C_DIS
LIN {X 58.093,Y -46.837,Z -171.251,A -90.000,B 90.000,C 0.000} C_DIS
LIN {X 57.970,Y -46.811,Z -172.453,A -90.000,B 90.000,C 0.000} C_DIS
LIN {X 57.972,Y -46.806,Z -172.577,A -90.000,B 90.000,C 0.000} C_DIS
LIN {X 57.967,Y -46.787,Z -173.205,A -90.000,B 90.000,C 0.000} C_DIS
LIN {X 57.963,Y -46.777,Z -173.786,A -90.000,B 90.000,C 0.000} C_DIS
LIN {X 57.955,Y -46.753,Z -174.550,A -90.000,B 90.000,C 0.000} C_DIS
LIN {X 58.297,Y -46.638,Z -176.253,A -90.000,B 90.000,C 0.000} C_DIS
LIN {X 58.336,Y -46.629,Z -176.450,A -90.000,B 90.000,C 0.000} C_DIS
LIN {X 58.372,Y -46.621,Z -176.570,A -90.000,B 90.000,C 0.000} C_DIS
LIN {X 58.425,Y -46.610,Z -176.761,A -90.000,B 90.000,C 0.000} C_DIS
LIN {X 58.450,Y -46.604,Z -176.867,A -90.000,B 90.000,C 0.000} C_DIS
LIN {X 58.474,Y -46.599,Z -176.979,A -90.000,B 90.000,C 0.000} C_DIS
LIN {X 58.552,Y -46.580,Z -177.407,A -90.000,B 90.000,C 0.000} C_DIS
LIN {X 58.581,Y -46.573,Z -177.601,A -90.000,B 90.000,C 0.000} C_DIS
LIN {X 58.596,Y -46.569,Z -177.722,A -90.000,B 90.000,C 0.000} C_DIS
LIN {X 58.692,Y -46.533,Z -178.856,A -90.000,B 90.000,C 0.000} C_DIS
LIN {X 58.710,Y -46.528,Z -179.117,A -90.000,B 90.000,C 0.000} C_DIS
LIN {X 58.734,Y -46.526,Z -179.885,A -90.000,B 90.000,C 0.000} C_DIS
LIN {X 58.752,Y -46.524,Z -179.981,A -90.000,B 90.000,C 0.000} C_DIS
LIN {X 58.778,Y -46.520,Z -180.136,A -90.000,B 90.000,C 0.000} C_DIS
LIN {X 58.814,Y -46.514,Z -180.383,A -90.000,B 90.000,C 0.000} C_DIS
LIN {X 58.882,Y -46.505,Z -180.958,A -90.000,B 90.000,C 0.000} C_DIS
LIN {X 59.004,Y -46.486,Z -182.014,A -90.000,B 90.000,C 0.000} C_DIS
LIN {X 59.115,Y -46.467,Z -182.459,A -90.000,B 90.000,C 0.000} C_DIS
LIN {X 59.173,Y -46.455,Z -182.693,A -90.000,B 90.000,C 0.000} C_DIS
LIN {X 59.584,Y -46.363,Z -184.361,A -90.000,B 90.000,C 0.000} C_DIS
LIN {X 59.624,Y -46.355,Z -184.542,A -90.000,B 90.000,C 0.000} C_DIS
LIN {X 59.664,Y -46.348,Z -184.760,A -90.000,B 90.000,C 0.000} C_DIS
LIN {X 59.691,Y -46.342,Z -184.920,A -90.000,B 90.000,C 0.000} C_DIS
LIN {X 59.721,Y -46.337,Z -185.139,A -90.000,B 90.000,C 0.000} C_DIS
LIN {X 59.740,Y -46.333,Z -185.310,A -90.000,B 90.000,C 0.000} C_DIS
LIN {X 59.761,Y -46.329,Z -185.556,A -90.000,B 90.000,C 0.000} C_DIS
LIN {X 59.773,Y -46.326,Z -185.754,A -90.000,B 90.000,C 0.000} C_DIS
LIN {X 59.789,Y -46.321,Z -186.342,A -90.000,B 90.000,C 0.000} C_DIS
LIN {X 59.839,Y -46.303,Z -188.353,A -90.000,B 90.000,C 0.000} C_DIS
LIN {X 59.850,Y -46.298,Z -188.927,A -90.000,B 90.000,C 0.000} C_DIS
LIN {X 59.861,Y -46.289,Z -189.596,A -90.000,B 90.000,C 0.000} C_DIS
LIN {X 59.863,Y -46.286,Z -189.798,A -90.000,B 90.000,C 0.000} C_DIS
LIN {X 59.822,Y -46.263,Z -191.632,A -90.000,B 90.000,C 0.000} C_DIS
LIN {X 59.795,Y -46.259,Z -192.137,A -90.000,B 90.000,C 0.000} C_DIS
LIN {X 59.758,Y -46.242,Z -192.755,A -90.000,B 90.000,C 0.000} C_DIS
LIN {X 59.641,Y -46.167,Z -194.533,A -90.000,B 90.000,C 0.000} C_DIS
LIN {X 59.554,Y -46.133,Z -195.481,A -90.000,B 90.000,C 0.000} C_DIS
LIN {X 59.543,Y -46.130,Z -195.571,A -90.000,B 90.000,C 0.000} C_DIS
LIN {X 59.498,Y -46.123,Z -195.895,A -90.000,B 90.000,C 0.000} C_DIS
LIN {X 59.440,Y -46.116,Z -196.228,A -90.000,B 90.000,C 0.000} C_DIS
LIN {X 59.397,Y -46.105,Z -196.529,A -90.000,B 90.000,C 0.000} C_DIS
LIN {X 59.266,Y -46.072,Z -197.424,A -90.000,B 90.000,C 0.000} C_DIS
LIN {X 59.221,Y -46.061,Z -197.719,A -90.000,B 90.000,C 0.000} C_DIS
LIN {X 59.165,Y -46.054,Z -198.013,A -90.000,B 90.000,C 0.000} C_DIS
LIN {X 59.134,Y -46.051,Z -198.159,A -90.000,B 90.000,C 0.000} C_DIS
LIN {X 58.708,Y -46.032,Z -199.889,A -90.000,B 90.000,C 0.000} C_DIS
LIN {X 58.606,Y -46.028,Z -200.290,A -90.000,B 90.000,C 0.000} C_DIS
LIN {X 57.613,Y -45.997,Z -203.693,A -90.000,B 90.000,C 0.000} C_DIS
LIN {X 57.289,Y -45.986,Z -204.802,A -90.000,B 90.000,C 0.000} C_DIS
LIN {X 57.096,Y -45.980,Z -205.418,A -90.000,B 90.000,C 0.000} C_DIS
LIN {X 55.862,Y -45.950,Z -209.259,A -90.000,B 90.000,C 0.000} C_DIS
LIN {X 54.987,Y -45.925,Z -211.920,A -90.000,B 90.000,C 0.000} C_DIS
LIN {X 54.182,Y -45.909,Z -214.288,A -90.000,B 90.000,C 0.000} C_DIS
LIN {X 53.389,Y -45.895,Z -216.561,A -90.000,B 90.000,C 0.000} C_DIS
LIN {X 52.370,Y -45.851,Z -219.638,A -90.000,B 90.000,C 0.000} C_DIS
LIN {X 52.322,Y -45.847,Z -219.780,A -90.000,B 90.000,C 0.000} C_DIS
LIN {X 52.202,Y -45.843,Z -220.099,A -90.000,B 90.000,C 0.000} C_DIS
LIN {X 51.995,Y -45.841,Z -220.596,A -90.000,B 90.000,C 0.000} C_DIS
LIN {X 51.699,Y -45.834,Z -221.301,A -90.000,B 90.000,C 0.000} C_DIS
LIN {X 50.245,Y -45.768,Z -224.972,A -90.000,B 90.000,C 0.000} C_DIS
LIN {X 50.075,Y -45.751,Z -225.389,A -90.000,B 90.000,C 0.000} C_DIS
LIN {X 50.042,Y -45.749,Z -225.466,A -90.000,B 90.000,C 0.000} C_DIS
LIN {X 49.977,Y -45.745,Z -225.610,A -90.000,B 90.000,C 0.000} C_DIS
LIN {X 49.870,Y -45.743,Z -225.827,A -90.000,B 90.000,C 0.000} C_DIS
LIN {X 49.828,Y -45.743,Z -225.908,A -90.000,B 90.000,C 0.000} C_DIS
LIN {X 49.491,Y -45.748,Z -226.523,A -90.000,B 90.000,C 0.000} C_DIS
LIN {X 48.274,Y -45.749,Z -228.844,A -90.000,B 90.000,C 0.000} C_DIS
LIN {X 47.721,Y -45.750,Z -229.901,A -90.000,B 90.000,C 0.000} C_DIS
LIN {X 47.559,Y -45.751,Z -230.209,A -90.000,B 90.000,C 0.000} C_DIS
LIN {X 47.448,Y -45.748,Z -230.420,A -90.000,B 90.000,C 0.000} C_DIS
LIN {X 47.070,Y -45.725,Z -231.122,A -90.000,B 90.000,C 0.000} C_DIS
LIN {X 47.017,Y -45.723,Z -231.214,A -90.000,B 90.000,C 0.000} C_DIS
LIN {X 46.874,Y -45.720,Z -231.454,A -90.000,B 90.000,C 0.000} C_DIS
LIN {X 46.741,Y -45.720,Z -231.661,A -90.000,B 90.000,C 0.000} C_DIS
LIN {X 46.568,Y -45.725,Z -231.911,A -90.000,B 90.000,C 0.000} C_DIS
LIN {X 46.435,Y -45.731,Z -232.092,A -90.000,B 90.000,C 0.000} C_DIS
LIN {X 45.983,Y -45.757,Z -232.677,A -90.000,B 90.000,C 0.000} C_DIS
LIN {X 43.910,Y -45.855,Z -235.463,A -90.000,B 90.000,C 0.000} C_DIS
LIN {X 43.610,Y -45.850,Z -235.858,A -90.000,B 90.000,C 0.000} C_DIS
LIN {X 42.816,Y -45.826,Z -236.897,A -90.000,B 90.000,C 0.000} C_DIS
LIN {X 42.679,Y -45.823,Z -237.068,A -90.000,B 90.000,C 0.000} C_DIS
LIN {X 42.583,Y -45.823,Z -237.178,A -90.000,B 90.000,C 0.000} C_DIS
LIN {X 42.327,Y -45.827,Z -237.452,A -90.000,B 90.000,C 0.000} C_DIS
LIN {X 42.161,Y -45.832,Z -237.618,A -90.000,B 90.000,C 0.000} C_DIS
LIN {X 41.827,Y -45.847,Z -237.927,A -90.000,B 90.000,C 0.000} C_DIS
LIN {X 41.493,Y -45.865,Z -238.215,A -90.000,B 90.000,C 0.000} C_DIS
LIN {X 39.300,Y -45.965,Z -240.092,A -90.000,B 90.000,C 0.000} C_DIS
LIN {X 38.620,Y -45.968,Z -240.663,A -90.000,B 90.000,C 0.000} C_DIS
LIN {X 37.516,Y -45.967,Z -241.617,A -90.000,B 90.000,C 0.000} C_DIS
LIN {X 36.879,Y -45.971,Z -242.170,A -90.000,B 90.000,C 0.000} C_DIS
LIN {X 36.815,Y -45.971,Z -242.223,A -90.000,B 90.000,C 0.000} C_DIS
LIN {X 36.601,Y -45.975,Z -242.396,A -90.000,B 90.000,C 0.000} C_DIS
LIN {X 36.248,Y -45.985,Z -242.662,A -90.000,B 90.000,C 0.000} C_DIS
LIN {X 35.973,Y -45.996,Z -242.855,A -90.000,B 90.000,C 0.000} C_DIS
LIN {X 35.146,Y -46.035,Z -243.399,A -90.000,B 90.000,C 0.000} C_DIS
LIN {X 34.891,Y -46.048,Z -243.561,A -90.000,B 90.000,C 0.000} C_DIS
LIN {X 34.033,Y -46.092,Z -244.113,A -90.000,B 90.000,C 0.000} C_DIS
LIN {X 33.794,Y -46.103,Z -244.270,A -90.000,B 90.000,C 0.000} C_DIS
LIN {X 33.670,Y -46.106,Z -244.358,A -90.000,B 90.000,C 0.000} C_DIS
LIN {X 33.647,Y -46.107,Z -244.375,A -90.000,B 90.000,C 0.000} C_DIS
LIN {X 33.646,Y -46.106,Z -244.379,A -90.000,B 90.000,C 0.000} C_DIS
LIN {X 33.728,Y -46.101,Z -244.339,A -90.000,B 90.000,C 0.000} C_DIS
LIN {X 33.894,Y -46.091,Z -244.245,A -90.000,B 90.000,C 0.000} C_DIS
LIN {X 36.254,Y -45.950,Z -242.843,A -90.000,B 90.000,C 0.000} C_DIS
LIN {X 37.356,Y -45.882,Z -242.198,A -90.000,B 90.000,C 0.000} C_DIS
LIN {X 37.927,Y -45.846,Z -241.868,A -90.000,B 90.000,C 0.000} C_DIS
LIN {X 39.065,Y -45.773,Z -241.221,A -90.000,B 90.000,C 0.000} C_DIS
LIN {X 39.615,Y -45.736,Z -240.915,A -90.000,B 90.000,C 0.000} C_DIS
LIN {X 40.141,Y -45.698,Z -240.629,A -90.000,B 90.000,C 0.000} C_DIS
LIN {X 40.393,Y -45.673,Z -240.495,A -90.000,B 90.000,C 0.000} C_DIS
LIN {X 40.635,Y -45.639,Z -240.368,A -90.000,B 90.000,C 0.000} C_DIS
LIN {X 40.867,Y -45.602,Z -240.249,A -90.000,B 90.000,C 0.000} C_DIS
LIN {X 41.295,Y -45.523,Z -240.036,A -90.000,B 90.000,C 0.000} C_DIS
LIN {X 41.489,Y -45.486,Z -239.945,A -90.000,B 90.000,C 0.000} C_DIS
LIN {X 41.752,Y -45.434,Z -239.827,A -90.000,B 90.000,C 0.000} C_DIS
LIN {X 41.908,Y -45.401,Z -239.763,A -90.000,B 90.000,C 0.000} C_DIS
LIN {X 42.047,Y -45.371,Z -239.711,A -90.000,B 90.000,C 0.000} C_DIS
LIN {X 42.168,Y -45.343,Z -239.672,A -90.000,B 90.000,C 0.000} C_DIS
LIN {X 42.269,Y -45.318,Z -239.646,A -90.000,B 90.000,C 0.000} C_DIS
LIN {X 42.350,Y -45.296,Z -239.635,A -90.000,B 90.000,C 0.000} C_DIS
LIN {X 42.396,Y -45.281,Z -239.637,A -90.000,B 90.000,C 0.000} C_DIS
LIN {X 42.420,Y -45.273,Z -239.642,A -90.000,B 90.000,C 0.000} C_DIS
LIN {X 42.436,Y -45.266,Z -239.651,A -90.000,B 90.000,C 0.000} C_DIS
LIN {X 42.443,Y -45.263,Z -239.658,A -90.000,B 90.000,C 0.000} C_DIS
LIN {X 42.451,Y -45.257,Z -239.673,A -90.000,B 90.000,C 0.000} C_DIS
LIN {X 42.452,Y -45.252,Z -239.692,A -90.000,B 90.000,C 0.000} C_DIS
LIN {X 42.448,Y -45.248,Z -239.715,A -90.000,B 90.000,C 0.000} C_DIS
LIN {X 42.436,Y -45.245,Z -239.744,A -90.000,B 90.000,C 0.000} C_DIS
LIN {X 42.394,Y -45.241,Z -239.817,A -90.000,B 90.000,C 0.000} C_DIS
LIN {X 42.326,Y -45.240,Z -239.909,A -90.000,B 90.000,C 0.000} C_DIS
LIN {X 42.229,Y -45.247,Z -240.019,A -90.000,B 90.000,C 0.000} C_DIS
LIN {X 42.032,Y -45.262,Z -240.223,A -90.000,B 90.000,C 0.000} C_DIS
LIN {X 41.861,Y -45.275,Z -240.386,A -90.000,B 90.000,C 0.000} C_DIS
LIN {X 41.659,Y -45.290,Z -240.571,A -90.000,B 90.000,C 0.000} C_DIS
LIN {X 41.424,Y -45.308,Z -240.779,A -90.000,B 90.000,C 0.000} C_DIS
LIN {X 41.221,Y -45.324,Z -240.955,A -90.000,B 90.000,C 0.000} C_DIS
LIN {X 39.874,Y -45.393,Z -242.112,A -90.000,B 90.000,C 0.000} C_DIS
LIN {X 38.787,Y -45.442,Z -243.070,A -90.000,B 90.000,C 0.000} C_DIS
LIN {X 38.223,Y -45.452,Z -243.561,A -90.000,B 90.000,C 0.000} C_DIS
LIN {X 38.223,Y -60.000,Z -243.561,A -90.000,B 90.000,C 0.000} C_DIS
LIN {X 11.684,Y -60.000,Z -243.561,A -90.000,B 90.000,C 0.000} C_DIS
LIN {X 11.684,Y -46.816,Z -243.561,A -90.000,B 90.000,C 0.000} C_DIS
LIN {X 11.454,Y -46.796,Z -243.173,A -90.000,B 90.000,C 0.000} C_DIS
LIN {X 10.257,Y -46.664,Z -241.138,A -90.000,B 90.000,C 0.000} C_DIS
LIN {X 10.063,Y -46.642,Z -240.790,A -90.000,B 90.000,C 0.000} C_DIS
LIN {X 9.914,Y -46.625,Z -240.500,A -90.000,B 90.000,C 0.000} C_DIS
LIN {X 9.802,Y -46.612,Z -240.262,A -90.000,B 90.000,C 0.000} C_DIS
LIN {X 9.693,Y -46.599,Z -240.006,A -90.000,B 90.000,C 0.000} C_DIS
LIN {X 9.660,Y -46.596,Z -239.924,A -90.000,B 90.000,C 0.000} C_DIS
LIN {X 9.576,Y -46.584,Z -239.687,A -90.000,B 90.000,C 0.000} C_DIS
LIN {X 9.489,Y -46.571,Z -239.412,A -90.000,B 90.000,C 0.000} C_DIS
LIN {X 9.404,Y -46.535,Z -239.132,A -90.000,B 90.000,C 0.000} C_DIS
LIN {X 9.340,Y -46.508,Z -238.906,A -90.000,B 90.000,C 0.000} C_DIS
LIN {X 9.284,Y -46.482,Z -238.677,A -90.000,B 90.000,C 0.000} C_DIS
LIN {X 9.234,Y -46.455,Z -238.429,A -90.000,B 90.000,C 0.000} C_DIS
LIN {X 9.202,Y -46.435,Z -238.237,A -90.000,B 90.000,C 0.000} C_DIS
LIN {X 9.111,Y -46.365,Z -237.533,A -90.000,B 90.000,C 0.000} C_DIS
LIN {X 9.077,Y -46.332,Z -237.176,A -90.000,B 90.000,C 0.000} C_DIS
LIN {X 9.062,Y -46.312,Z -236.960,A -90.000,B 90.000,C 0.000} C_DIS
LIN {X 9.049,Y -46.284,Z -236.639,A -90.000,B 90.000,C 0.000} C_DIS
LIN {X 9.046,Y -46.268,Z -236.450,A -90.000,B 90.000,C 0.000} C_DIS
LIN {X 9.048,Y -46.248,Z -236.198,A -90.000,B 90.000,C 0.000} C_DIS
LIN {X 9.061,Y -46.223,Z -235.874,A -90.000,B 90.000,C 0.000} C_DIS
LIN {X 9.083,Y -46.205,Z -235.611,A -90.000,B 90.000,C 0.000} C_DIS
LIN {X 9.106,Y -46.192,Z -235.411,A -90.000,B 90.000,C 0.000} C_DIS
LIN {X 9.133,Y -46.179,Z -235.210,A -90.000,B 90.000,C 0.000} C_DIS
LIN {X 9.188,Y -46.160,Z -234.889,A -90.000,B 90.000,C 0.000} C_DIS
LIN {X 9.424,Y -46.098,Z -233.735,A -90.000,B 90.000,C 0.000} C_DIS
LIN {X 9.491,Y -46.075,Z -233.411,A -90.000,B 90.000,C 0.000} C_DIS
LIN {X 9.617,Y -46.042,Z -232.797,A -90.000,B 90.000,C 0.000} C_DIS
LIN {X 9.977,Y -45.899,Z -231.092,A -90.000,B 90.000,C 0.000} C_DIS
LIN {X 10.240,Y -45.795,Z -229.851,A -90.000,B 90.000,C 0.000} C_DIS
LIN {X 10.361,Y -45.756,Z -229.357,A -90.000,B 90.000,C 0.000} C_DIS
LIN {X 10.460,Y -45.733,Z -229.016,A -90.000,B 90.000,C 0.000} C_DIS
LIN {X 11.421,Y -45.558,Z -226.051,A -90.000,B 90.000,C 0.000} C_DIS
LIN {X 11.969,Y -45.459,Z -224.373,A -90.000,B 90.000,C 0.000} C_DIS
LIN {X 12.055,Y -45.445,Z -224.133,A -90.000,B 90.000,C 0.000} C_DIS
LIN {X 12.162,Y -45.432,Z -223.862,A -90.000,B 90.000,C 0.000} C_DIS
LIN {X 12.540,Y -45.396,Z -222.994,A -90.000,B 90.000,C 0.000} C_DIS
LIN {X 12.652,Y -45.389,Z -222.743,A -90.000,B 90.000,C 0.000} C_DIS
LIN {X 13.480,Y -45.358,Z -221.045,A -90.000,B 90.000,C 0.000} C_DIS
LIN {X 14.001,Y -45.347,Z -220.039,A -90.000,B 90.000,C 0.000} C_DIS
LIN {X 14.865,Y -45.322,Z -218.377,A -90.000,B 90.000,C 0.000} C_DIS
LIN {X 15.358,Y -45.319,Z -217.423,A -90.000,B 90.000,C 0.000} C_DIS
LIN {X 15.796,Y -45.324,Z -216.619,A -90.000,B 90.000,C 0.000} C_DIS
LIN {X 17.313,Y -45.350,Z -213.834,A -90.000,B 90.000,C 0.000} C_DIS
LIN {X 17.784,Y -45.355,Z -212.897,A -90.000,B 90.000,C 0.000} C_DIS
LIN {X 17.975,Y -45.363,Z -212.518,A -90.000,B 90.000,C 0.000} C_DIS
LIN {X 19.560,Y -45.451,Z -209.636,A -90.000,B 90.000,C 0.000} C_DIS
LIN {X 19.717,Y -45.455,Z -209.302,A -90.000,B 90.000,C 0.000} C_DIS
LIN {X 19.870,Y -45.463,Z -208.974,A -90.000,B 90.000,C 0.000} C_DIS
LIN {X 20.293,Y -45.489,Z -208.065,A -90.000,B 90.000,C 0.000} C_DIS
LIN {X 20.454,Y -45.500,Z -207.741,A -90.000,B 90.000,C 0.000} C_DIS
LIN {X 21.271,Y -45.570,Z -206.232,A -90.000,B 90.000,C 0.000} C_DIS
LIN {X 21.408,Y -45.576,Z -205.907,A -90.000,B 90.000,C 0.000} C_DIS
LIN {X 21.791,Y -45.600,Z -204.993,A -90.000,B 90.000,C 0.000} C_DIS
LIN {X 22.252,Y -45.640,Z -203.888,A -90.000,B 90.000,C 0.000} C_DIS
LIN {X 22.357,Y -45.649,Z -203.641,A -90.000,B 90.000,C 0.000} C_DIS
LIN {X 22.492,Y -45.663,Z -203.353,A -90.000,B 90.000,C 0.000} C_DIS
LIN {X 22.721,Y -45.688,Z -202.904,A -90.000,B 90.000,C 0.000} C_DIS
LIN {X 22.907,Y -45.706,Z -202.364,A -90.000,B 90.000,C 0.000} C_DIS
LIN {X 23.462,Y -45.762,Z -200.759,A -90.000,B 90.000,C 0.000} C_DIS
LIN {X 23.557,Y -45.770,Z -200.502,A -90.000,B 90.000,C 0.000} C_DIS
LIN {X 23.848,Y -45.801,Z -199.785,A -90.000,B 90.000,C 0.000} C_DIS
LIN {X 23.884,Y -45.806,Z -199.676,A -90.000,B 90.000,C 0.000} C_DIS
LIN {X 24.851,Y -45.939,Z -197.135,A -90.000,B 90.000,C 0.000} C_DIS
LIN {X 24.869,Y -45.940,Z -197.030,A -90.000,B 90.000,C 0.000} C_DIS
LIN {X 24.890,Y -45.941,Z -196.923,A -90.000,B 90.000,C 0.000} C_DIS
LIN {X 24.949,Y -45.941,Z -196.644,A -90.000,B 90.000,C 0.000} C_DIS
LIN {X 25.007,Y -45.941,Z -196.411,A -90.000,B 90.000,C 0.000} C_DIS
LIN {X 25.051,Y -45.943,Z -196.244,A -90.000,B 90.000,C 0.000} C_DIS
LIN {X 25.160,Y -45.948,Z -195.874,A -90.000,B 90.000,C 0.000} C_DIS
LIN {X 25.258,Y -45.955,Z -195.581,A -90.000,B 90.000,C 0.000} C_DIS
LIN {X 25.754,Y -46.000,Z -194.248,A -90.000,B 90.000,C 0.000} C_DIS
LIN {X 25.842,Y -45.985,Z -193.600,A -90.000,B 90.000,C 0.000} C_DIS
LIN {X 25.894,Y -45.980,Z -193.279,A -90.000,B 90.000,C 0.000} C_DIS
LIN {X 25.948,Y -45.978,Z -193.005,A -90.000,B 90.000,C 0.000} C_DIS
LIN {X 26.018,Y -45.974,Z -192.698,A -90.000,B 90.000,C 0.000} C_DIS
LIN {X 26.079,Y -45.968,Z -192.463,A -90.000,B 90.000,C 0.000} C_DIS
LIN {X 26.150,Y -45.964,Z -192.223,A -90.000,B 90.000,C 0.000} C_DIS
LIN {X 26.202,Y -45.961,Z -192.056,A -90.000,B 90.000,C 0.000} C_DIS
LIN {X 26.346,Y -45.960,Z -191.652,A -90.000,B 90.000,C 0.000} C_DIS
LIN {X 26.429,Y -45.961,Z -191.438,A -90.000,B 90.000,C 0.000} C_DIS
LIN {X 26.719,Y -45.971,Z -190.767,A -90.000,B 90.000,C 0.000} C_DIS
LIN {X 26.883,Y -45.953,Z -190.116,A -90.000,B 90.000,C 0.000} C_DIS
LIN {X 27.117,Y -45.930,Z -189.188,A -90.000,B 90.000,C 0.000} C_DIS
LIN {X 27.158,Y -45.920,Z -189.034,A -90.000,B 90.000,C 0.000} C_DIS
LIN {X 27.261,Y -45.898,Z -188.693,A -90.000,B 90.000,C 0.000} C_DIS
LIN {X 27.335,Y -45.884,Z -188.478,A -90.000,B 90.000,C 0.000} C_DIS
LIN {X 27.375,Y -45.878,Z -188.372,A -90.000,B 90.000,C 0.000} C_DIS
LIN {X 27.458,Y -45.868,Z -188.170,A -90.000,B 90.000,C 0.000} C_DIS
LIN {X 27.583,Y -45.855,Z -187.884,A -90.000,B 90.000,C 0.000} C_DIS
LIN {X 27.656,Y -45.848,Z -187.722,A -90.000,B 90.000,C 0.000} C_DIS
LIN {X 27.790,Y -45.840,Z -187.447,A -90.000,B 90.000,C 0.000} C_DIS
LIN {X 27.940,Y -45.834,Z -187.165,A -90.000,B 90.000,C 0.000} C_DIS
LIN {X 28.064,Y -45.832,Z -186.947,A -90.000,B 90.000,C 0.000} C_DIS
LIN {X 28.682,Y -45.832,Z -185.936,A -90.000,B 90.000,C 0.000} C_DIS
LIN {X 29.156,Y -45.807,Z -185.173,A -90.000,B 90.000,C 0.000} C_DIS
LIN {X 29.477,Y -45.787,Z -184.655,A -90.000,B 90.000,C 0.000} C_DIS
LIN {X 30.046,Y -45.755,Z -183.775,A -90.000,B 90.000,C 0.000} C_DIS
LIN {X 30.208,Y -45.749,Z -183.538,A -90.000,B 90.000,C 0.000} C_DIS
LIN {X 30.316,Y -45.747,Z -183.390,A -90.000,B 90.000,C 0.000} C_DIS
LIN {X 30.611,Y -45.745,Z -183.013,A -90.000,B 90.000,C 0.000} C_DIS
LIN {X 30.789,Y -45.745,Z -182.800,A -90.000,B 90.000,C 0.000} C_DIS
LIN {X 30.940,Y -45.747,Z -182.629,A -90.000,B 90.000,C 0.000} C_DIS
LIN {X 31.894,Y -45.774,Z -181.619,A -90.000,B 90.000,C 0.000} C_DIS
LIN {X 32.553,Y -45.758,Z -180.790,A -90.000,B 90.000,C 0.000} C_DIS
LIN {X 32.763,Y -45.757,Z -180.528,A -90.000,B 90.000,C 0.000} C_DIS
LIN {X 32.972,Y -45.759,Z -180.284,A -90.000,B 90.000,C 0.000} C_DIS
LIN {X 33.155,Y -45.764,Z -180.081,A -90.000,B 90.000,C 0.000} C_DIS
LIN {X 33.410,Y -45.774,Z -179.815,A -90.000,B 90.000,C 0.000} C_DIS
LIN {X 33.551,Y -45.780,Z -179.675,A -90.000,B 90.000,C 0.000} C_DIS
LIN {X 33.733,Y -45.787,Z -179.505,A -90.000,B 90.000,C 0.000} C_DIS
LIN {X 34.334,Y -45.779,Z -178.777,A -90.000,B 90.000,C 0.000} C_DIS
LIN {X 34.679,Y -45.786,Z -178.353,A -90.000,B 90.000,C 0.000} C_DIS
LIN {X 34.971,Y -45.792,Z -178.018,A -90.000,B 90.000,C 0.000} C_DIS
LIN {X 35.225,Y -45.802,Z -177.748,A -90.000,B 90.000,C 0.000} C_DIS
LIN {X 35.522,Y -45.817,Z -177.454,A -90.000,B 90.000,C 0.000} C_DIS
LIN {X 35.749,Y -45.830,Z -177.237,A -90.000,B 90.000,C 0.000} C_DIS
LIN {X 36.673,Y -45.907,Z -176.346,A -90.000,B 90.000,C 0.000} C_DIS
LIN {X 36.879,Y -45.917,Z -176.094,A -90.000,B 90.000,C 0.000} C_DIS
LIN {X 37.111,Y -45.927,Z -175.806,A -90.000,B 90.000,C 0.000} C_DIS
LIN {X 37.504,Y -45.953,Z -175.313,A -90.000,B 90.000,C 0.000} C_DIS
LIN {X 38.014,Y -45.976,Z -174.604,A -90.000,B 90.000,C 0.000} C_DIS
LIN {X 38.209,Y -45.987,Z -174.331,A -90.000,B 90.000,C 0.000} C_DIS
LIN {X 38.449,Y -45.999,Z -173.974,A -90.000,B 90.000,C 0.000} C_DIS
LIN {X 39.543,Y -46.043,Z -172.281,A -90.000,B 90.000,C 0.000} C_DIS
LIN {X 40.034,Y -46.054,Z -171.454,A -90.000,B 90.000,C 0.000} C_DIS
LIN {X 40.760,Y -46.064,Z -170.274,A -90.000,B 90.000,C 0.000} C_DIS
LIN {X 41.155,Y -46.073,Z -169.588,A -90.000,B 90.000,C 0.000} C_DIS
LIN {X 41.369,Y -46.079,Z -169.243,A -90.000,B 90.000,C 0.000} C_DIS
LIN {X 41.439,Y -46.081,Z -169.134,A -90.000,B 90.000,C 0.000} C_DIS
LIN {X 41.588,Y -46.086,Z -168.916,A -90.000,B 90.000,C 0.000} C_DIS
LIN {X 41.774,Y -46.096,Z -168.664,A -90.000,B 90.000,C 0.000} C_DIS
LIN {X 41.969,Y -46.108,Z -168.415,A -90.000,B 90.000,C 0.000} C_DIS
LIN {X 42.028,Y -46.113,Z -168.342,A -90.000,B 90.000,C 0.000} C_DIS
LIN {X 42.167,Y -46.124,Z -168.182,A -90.000,B 90.000,C 0.000} C_DIS
LIN {X 42.374,Y -46.142,Z -167.956,A -90.000,B 90.000,C 0.000} C_DIS
LIN {X 42.456,Y -46.150,Z -167.873,A -90.000,B 90.000,C 0.000} C_DIS
LIN {X 42.691,Y -46.174,Z -167.641,A -90.000,B 90.000,C 0.000} C_DIS
LIN {X 42.802,Y -46.186,Z -167.537,A -90.000,B 90.000,C 0.000} C_DIS
LIN {X 42.906,Y -46.198,Z -167.444,A -90.000,B 90.000,C 0.000} C_DIS
LIN {X 43.154,Y -46.228,Z -167.236,A -90.000,B 90.000,C 0.000} C_DIS
LIN {X 43.336,Y -46.252,Z -167.093,A -90.000,B 90.000,C 0.000} C_DIS
LIN {X 43.509,Y -46.277,Z -166.963,A -90.000,B 90.000,C 0.000} C_DIS
LIN {X 43.735,Y -46.310,Z -166.805,A -90.000,B 90.000,C 0.000} C_DIS
LIN {X 44.144,Y -46.373,Z -166.540,A -90.000,B 90.000,C 0.000} C_DIS
LIN {X 44.982,Y -46.469,Z -166.004,A -90.000,B 90.000,C 0.000} C_DIS
LIN {X 45.710,Y -46.548,Z -165.505,A -90.000,B 90.000,C 0.000} C_DIS
LIN {X 45.851,Y -46.555,Z -165.333,A -90.000,B 90.000,C 0.000} C_DIS
LIN {X 46.021,Y -46.565,Z -165.138,A -90.000,B 90.000,C 0.000} C_DIS
LIN {X 46.267,Y -46.582,Z -164.878,A -90.000,B 90.000,C 0.000} C_DIS
LIN {X 46.369,Y -46.590,Z -164.778,A -90.000,B 90.000,C 0.000} C_DIS
LIN {X 46.576,Y -46.607,Z -164.587,A -90.000,B 90.000,C 0.000} C_DIS
LIN {X 46.886,Y -46.635,Z -164.322,A -90.000,B 90.000,C 0.000} C_DIS
LIN {X 47.160,Y -46.663,Z -164.099,A -90.000,B 90.000,C 0.000} C_DIS
LIN {X 47.290,Y -46.677,Z -164.004,A -90.000,B 90.000,C 0.000} C_DIS
LIN {X 47.526,Y -46.702,Z -163.836,A -90.000,B 90.000,C 0.000} C_DIS
LIN {X 47.683,Y -46.718,Z -163.728,A -90.000,B 90.000,C 0.000} C_DIS
LIN {X 47.831,Y -46.733,Z -163.631,A -90.000,B 90.000,C 0.000} C_DIS
LIN {X 48.127,Y -46.765,Z -163.452,A -90.000,B 90.000,C 0.000} C_DIS
LIN {X 48.293,Y -46.779,Z -163.358,A -90.000,B 90.000,C 0.000} C_DIS
LIN {X 48.609,Y -46.804,Z -163.195,A -90.000,B 90.000,C 0.000} C_DIS
LIN {X 49.028,Y -46.840,Z -163.007,A -90.000,B 90.000,C 0.000} C_DIS
LIN {X 49.263,Y -46.861,Z -162.911,A -90.000,B 90.000,C 0.000} C_DIS
LIN {X 49.416,Y -46.875,Z -162.854,A -90.000,B 90.000,C 0.000} C_DIS
LIN {X 49.661,Y -46.898,Z -162.771,A -90.000,B 90.000,C 0.000} C_DIS
LIN {X 49.784,Y -46.910,Z -162.732,A -90.000,B 90.000,C 0.000} C_DIS
LIN {X 50.042,Y -46.936,Z -162.659,A -90.000,B 90.000,C 0.000} C_DIS
LIN {X 50.337,Y -46.964,Z -162.586,A -90.000,B 90.000,C 0.000} C_DIS
LIN {X 50.550,Y -46.984,Z -162.543,A -90.000,B 90.000,C 0.000} C_DIS
LIN {X 50.780,Y -47.007,Z -162.505,A -90.000,B 90.000,C 0.000} C_DIS
LIN {X 51.062,Y -47.035,Z -162.465,A -90.000,B 90.000,C 0.000} C_DIS
LIN {X 51.390,Y -47.055,Z -162.424,A -90.000,B 90.000,C 0.000} C_DIS
LIN {X 51.582,Y -47.067,Z -162.408,A -90.000,B 90.000,C 0.000} C_DIS
LIN {X 51.717,Y -47.071,Z -162.399,A -90.000,B 90.000,C 0.000} C_DIS
LIN {X 52.008,Y -47.080,Z -162.391,A -90.000,B 90.000,C 0.000} C_DIS
LIN {X 52.253,Y -47.092,Z -162.393,A -90.000,B 90.000,C 0.000} C_DIS
LIN {X 52.518,Y -47.104,Z -162.403,A -90.000,B 90.000,C 0.000} C_DIS
LIN {X 52.696,Y -47.113,Z -162.416,A -90.000,B 90.000,C 0.000} C_DIS
LIN {X 52.887,Y -47.122,Z -162.434,A -90.000,B 90.000,C 0.000} C_DIS
LIN {X 53.089,Y -47.132,Z -162.456,A -90.000,B 90.000,C 0.000} C_DIS
LIN {X 53.434,Y -47.150,Z -162.508,A -90.000,B 90.000,C 0.000} C_DIS
LIN {X 53.639,Y -47.160,Z -162.546,A -90.000,B 90.000,C 0.000} C_DIS
LIN {X 53.881,Y -47.173,Z -162.599,A -90.000,B 90.000,C 0.000} C_DIS
LIN {X 54.258,Y -47.194,Z -162.696,A -90.000,B 90.000,C 0.000} C_DIS
LIN {X 54.360,Y -47.196,Z -162.726,A -90.000,B 90.000,C 0.000} C_DIS
LIN {X 54.494,Y -47.196,Z -162.767,A -90.000,B 90.000,C 0.000} C_DIS
LIN {X 54.729,Y -47.188,Z -162.846,A -90.000,B 90.000,C 0.000} C_DIS
LIN {X 54.916,Y -47.183,Z -162.916,A -90.000,B 90.000,C 0.000} C_DIS
LIN {X 55.192,Y -47.176,Z -163.026,A -90.000,B 90.000,C 0.000} C_DIS
LIN {X 55.289,Y -47.173,Z -163.068,A -90.000,B 90.000,C 0.000} C_DIS
LIN {X 55.517,Y -47.168,Z -163.174,A -90.000,B 90.000,C 0.000} C_DIS
LIN {X 55.781,Y -47.161,Z -163.306,A -90.000,B 90.000,C 0.000} C_DIS
LIN {X 55.959,Y -47.157,Z -163.403,A -90.000,B 90.000,C 0.000} C_DIS
LIN {X 56.163,Y -47.152,Z -163.523,A -90.000,B 90.000,C 0.000} C_DIS
LIN {X 56.408,Y -47.146,Z -163.674,A -90.000,B 90.000,C 0.000} C_DIS
LIN {X 56.607,Y -47.141,Z -163.806,A -90.000,B 90.000,C 0.000} C_DIS
LIN {X 56.819,Y -47.136,Z -163.958,A -90.000,B 90.000,C 0.000} C_DIS
LIN {X 57.039,Y -47.131,Z -164.127,A -90.000,B 90.000,C 0.000} C_DIS
LIN {X 57.140,Y -47.128,Z -164.209,A -90.000,B 90.000,C 0.000} C_DIS
LIN {X 57.287,Y -47.114,Z -164.333,A -90.000,B 90.000,C 0.000} C_DIS
LIN {X 57.435,Y -47.100,Z -164.466,A -90.000,B 90.000,C 0.000} C_DIS
LIN {X 57.645,Y -47.076,Z -164.663,A -90.000,B 90.000,C 0.000} C_DIS
LIN {X 57.799,Y -47.057,Z -164.818,A -90.000,B 90.000,C 0.000} C_DIS
LIN {X 58.031,Y -47.028,Z -165.071,A -90.000,B 90.000,C 0.000} C_DIS
LIN {X 58.249,Y -47.001,Z -165.325,A -90.000,B 90.000,C 0.000} C_DIS
LIN {X 58.493,Y -46.969,Z -165.642,A -90.000,B 90.000,C 0.000} C_DIS
LIN {X 58.707,Y -46.941,Z -165.948,A -90.000,B 90.000,C 0.000} C_DIS
LIN {X 58.770,Y -46.932,Z -166.045,A -90.000,B 90.000,C 0.000} C_DIS
LIN {X 58.943,Y -46.908,Z -166.329,A -90.000,B 90.000,C 0.000} C_DIS
LIN {X 59.029,Y -46.896,Z -166.480,A -90.000,B 90.000,C 0.000} C_DIS
LIN {X 59.152,Y -46.879,Z -166.710,A -90.000,B 90.000,C 0.000} C_DIS
LIN {X 59.250,Y -46.865,Z -166.910,A -90.000,B 90.000,C 0.000} C_DIS
LIN {X 59.308,Y -46.855,Z -167.035,A -90.000,B 90.000,C 0.000} C_DIS
LIN {X 59.416,Y -46.836,Z -167.278,A -90.000,B 90.000,C 0.000} C_DIS
LIN {X 59.467,Y -46.826,Z -167.403,A -90.000,B 90.000,C 0.000} C_DIS
LIN {X 59.603,Y -46.800,Z -167.769,A -90.000,B 90.000,C 0.000} C_DIS
LIN {X 59.717,Y -46.777,Z -168.108,A -90.000,B 90.000,C 0.000} C_DIS
LIN {X 59.789,Y -46.752,Z -168.348,A -90.000,B 90.000,C 0.000} C_DIS
LIN {X 59.882,Y -46.717,Z -168.699,A -90.000,B 90.000,C 0.000} C_DIS
LIN {X 59.944,Y -46.692,Z -168.974,A -90.000,B 90.000,C 0.000} C_DIS
LIN {X 59.963,Y -46.683,Z -169.078,A -90.000,B 90.000,C 0.000} C_DIS
LIN {X 59.994,Y -46.668,Z -169.258,A -90.000,B 90.000,C 0.000} C_DIS
LIN {X 60.031,Y -46.645,Z -169.551,A -90.000,B 90.000,C 0.000} C_DIS
LIN {X 60.040,Y -46.639,Z -169.645,A -90.000,B 90.000,C 0.000} C_DIS
LIN {X 60.089,Y -46.599,Z -170.219,A -90.000,B 90.000,C 0.000} C_DIS
LIN {X 60.098,Y -46.587,Z -170.410,A -90.000,B 90.000,C 0.000} C_DIS
LIN {X 60.101,Y -46.565,Z -170.805,A -90.000,B 90.000,C 0.000} C_DIS
LIN {X 60.094,Y -46.554,Z -171.032,A -90.000,B 90.000,C 0.000} C_DIS
LIN {X 60.089,Y -46.550,Z -171.121,A -90.000,B 90.000,C 0.000} C_DIS
LIN {X 60.065,Y -46.539,Z -171.402,A -90.000,B 90.000,C 0.000} C_DIS
LIN {X 59.948,Y -46.499,Z -172.534,A -90.000,B 90.000,C 0.000} C_DIS
LIN {X 59.936,Y -46.448,Z -173.580,A -90.000,B 90.000,C 0.000} C_DIS
LIN {X 59.929,Y -46.425,Z -174.347,A -90.000,B 90.000,C 0.000} C_DIS
LIN {X 60.251,Y -46.318,Z -175.955,A -90.000,B 90.000,C 0.000} C_DIS
LIN {X 60.325,Y -46.297,Z -176.222,A -90.000,B 90.000,C 0.000} C_DIS
LIN {X 60.366,Y -46.285,Z -176.389,A -90.000,B 90.000,C 0.000} C_DIS
LIN {X 60.412,Y -46.270,Z -176.614,A -90.000,B 90.000,C 0.000} C_DIS
LIN {X 60.490,Y -46.250,Z -177.039,A -90.000,B 90.000,C 0.000} C_DIS
LIN {X 60.529,Y -46.239,Z -177.289,A -90.000,B 90.000,C 0.000} C_DIS
LIN {X 60.553,Y -46.230,Z -177.494,A -90.000,B 90.000,C 0.000} C_DIS
LIN {X 60.605,Y -46.210,Z -178.090,A -90.000,B 90.000,C 0.000} C_DIS
LIN {X 60.654,Y -46.184,Z -178.678,A -90.000,B 90.000,C 0.000} C_DIS
LIN {X 60.673,Y -46.172,Z -178.979,A -90.000,B 90.000,C 0.000} C_DIS
LIN {X 60.684,Y -46.160,Z -179.355,A -90.000,B 90.000,C 0.000} C_DIS
LIN {X 60.693,Y -46.156,Z -179.674,A -90.000,B 90.000,C 0.000} C_DIS
LIN {X 60.714,Y -46.150,Z -179.794,A -90.000,B 90.000,C 0.000} C_DIS
LIN {X 60.757,Y -46.138,Z -180.092,A -90.000,B 90.000,C 0.000} C_DIS
LIN {X 60.933,Y -46.082,Z -181.651,A -90.000,B 90.000,C 0.000} C_DIS
LIN {X 61.011,Y -46.062,Z -181.966,A -90.000,B 90.000,C 0.000} C_DIS
LIN {X 61.497,Y -45.962,Z -183.936,A -90.000,B 90.000,C 0.000} C_DIS
LIN {X 61.534,Y -45.955,Z -184.108,A -90.000,B 90.000,C 0.000} C_DIS
LIN {X 61.587,Y -45.943,Z -184.391,A -90.000,B 90.000,C 0.000} C_DIS
LIN {X 61.619,Y -45.935,Z -184.580,A -90.000,B 90.000,C 0.000} C_DIS
LIN {X 61.666,Y -45.926,Z -184.918,A -90.000,B 90.000,C 0.000} C_DIS
LIN {X 61.682,Y -45.923,Z -185.060,A -90.000,B 90.000,C 0.000} C_DIS
LIN {X 61.711,Y -45.917,Z -185.386,A -90.000,B 90.000,C 0.000} C_DIS
LIN {X 61.726,Y -45.915,Z -185.630,A -90.000,B 90.000,C 0.000} C_DIS
LIN {X 61.746,Y -45.913,Z -186.328,A -90.000,B 90.000,C 0.000} C_DIS
LIN {X 61.768,Y -45.889,Z -187.323,A -90.000,B 90.000,C 0.000} C_DIS
LIN {X 61.788,Y -45.857,Z -188.312,A -90.000,B 90.000,C 0.000} C_DIS
LIN {X 61.804,Y -45.817,Z -189.574,A -90.000,B 90.000,C 0.000} C_DIS
LIN {X 61.805,Y -45.811,Z -189.776,A -90.000,B 90.000,C 0.000} C_DIS
LIN {X 61.796,Y -45.802,Z -190.189,A -90.000,B 90.000,C 0.000} C_DIS
LIN {X 61.752,Y -45.747,Z -191.726,A -90.000,B 90.000,C 0.000} C_DIS
LIN {X 61.668,Y -45.709,Z -193.118,A -90.000,B 90.000,C 0.000} C_DIS
LIN {X 61.568,Y -45.644,Z -194.637,A -90.000,B 90.000,C 0.000} C_DIS
LIN {X 61.477,Y -45.608,Z -195.637,A -90.000,B 90.000,C 0.000} C_DIS
LIN {X 61.462,Y -45.604,Z -195.776,A -90.000,B 90.000,C 0.000} C_DIS
LIN {X 61.410,Y -45.595,Z -196.152,A -90.000,B 90.000,C 0.000} C_DIS
LIN {X 61.356,Y -45.590,Z -196.473,A -90.000,B 90.000,C 0.000} C_DIS
LIN {X 61.264,Y -45.568,Z -197.091,A -90.000,B 90.000,C 0.000} C_DIS
LIN {X 61.131,Y -45.535,Z -197.991,A -90.000,B 90.000,C 0.000} C_DIS
LIN {X 61.063,Y -45.525,Z -198.359,A -90.000,B 90.000,C 0.000} C_DIS
LIN {X 61.007,Y -45.520,Z -198.617,A -90.000,B 90.000,C 0.000} C_DIS
LIN {X 60.582,Y -45.502,Z -200.344,A -90.000,B 90.000,C 0.000} C_DIS
LIN {X 60.517,Y -45.499,Z -200.599,A -90.000,B 90.000,C 0.000} C_DIS
LIN {X 60.458,Y -45.495,Z -200.824,A -90.000,B 90.000,C 0.000} C_DIS
LIN {X 59.396,Y -45.454,Z -204.457,A -90.000,B 90.000,C 0.000} C_DIS
LIN {X 59.135,Y -45.434,Z -205.336,A -90.000,B 90.000,C 0.000} C_DIS
LIN {X 58.930,Y -45.420,Z -205.986,A -90.000,B 90.000,C 0.000} C_DIS
LIN {X 57.676,Y -45.350,Z -209.850,A -90.000,B 90.000,C 0.000} C_DIS
LIN {X 57.023,Y -45.308,Z -211.810,A -90.000,B 90.000,C 0.000} C_DIS
LIN {X 57.023,Y -60.000,Z -211.810,A -90.000,B 90.000,C 0.000} C_DIS
LIN {X 35.139,Y -60.000,Z -175.166,A -90.000,B 90.000,C 0.000} C_DIS
LIN {X 35.139,Y -45.308,Z -175.166,A -90.000,B 90.000,C 0.000} C_DIS
LIN {X 35.282,Y -45.326,Z -175.026,A -90.000,B 90.000,C 0.000} C_DIS
LIN {X 35.544,Y -45.346,Z -174.699,A -90.000,B 90.000,C 0.000} C_DIS
LIN {X 36.000,Y -45.375,Z -174.127,A -90.000,B 90.000,C 0.000} C_DIS
LIN {X 36.555,Y -45.413,Z -173.348,A -90.000,B 90.000,C 0.000} C_DIS
LIN {X 36.645,Y -45.417,Z -173.223,A -90.000,B 90.000,C 0.000} C_DIS
LIN {X 36.858,Y -45.423,Z -172.908,A -90.000,B 90.000,C 0.000} C_DIS
LIN {X 37.367,Y -45.433,Z -172.127,A -90.000,B 90.000,C 0.000} C_DIS
LIN {X 37.602,Y -45.442,Z -171.763,A -90.000,B 90.000,C 0.000} C_DIS
LIN {X 37.924,Y -45.451,Z -171.266,A -90.000,B 90.000,C 0.000} C_DIS
LIN {X 38.411,Y -45.455,Z -170.450,A -90.000,B 90.000,C 0.000} C_DIS
LIN {X 38.659,Y -45.460,Z -170.045,A -90.000,B 90.000,C 0.000} C_DIS
LIN {X 39.127,Y -45.478,Z -169.278,A -90.000,B 90.000,C 0.000} C_DIS
LIN {X 39.503,Y -45.486,Z -168.627,A -90.000,B 90.000,C 0.000} C_DIS
LIN {X 39.765,Y -45.496,Z -168.201,A -90.000,B 90.000,C 0.000} C_DIS
LIN {X 39.871,Y -45.502,Z -168.037,A -90.000,B 90.000,C 0.000} C_DIS
LIN {X 40.023,Y -45.510,Z -167.813,A -90.000,B 90.000,C 0.000} C_DIS
LIN {X 40.277,Y -45.527,Z -167.466,A -90.000,B 90.000,C 0.000} C_DIS
LIN {X 40.471,Y -45.542,Z -167.216,A -90.000,B 90.000,C 0.000} C_DIS
LIN {X 40.550,Y -45.550,Z -167.119,A -90.000,B 90.000,C 0.000} C_DIS
LIN {X 40.775,Y -45.572,Z -166.855,A -90.000,B 90.000,C 0.000} C_DIS
LIN {X 40.979,Y -45.596,Z -166.631,A -90.000,B 90.000,C 0.000} C_DIS
LIN {X 41.109,Y -45.613,Z -166.495,A -90.000,B 90.000,C 0.000} C_DIS
LIN {X 41.400,Y -45.655,Z -166.204,A -90.000,B 90.000,C 0.000} C_DIS
LIN {X 41.566,Y -45.681,Z -166.048,A -90.000,B 90.000,C 0.000} C_DIS
LIN {X 41.705,Y -45.702,Z -165.924,A -90.000,B 90.000,C 0.000} C_DIS
LIN {X 41.996,Y -45.741,Z -165.680,A -90.000,B 90.000,C 0.000} C_DIS
LIN {X 42.178,Y -45.766,Z -165.536,A -90.000,B 90.000,C 0.000} C_DIS
LIN {X 42.409,Y -45.800,Z -165.362,A -90.000,B 90.000,C 0.000} C_DIS
LIN {X 42.702,Y -45.845,Z -165.157,A -90.000,B 90.000,C 0.000} C_DIS
LIN {X 43.938,Y -46.041,Z -164.352,A -90.000,B 90.000,C 0.000} C_DIS
LIN {X 44.399,Y -46.111,Z -164.032,A -90.000,B 90.000,C 0.000} C_DIS
LIN {X 44.563,Y -46.125,Z -163.842,A -90.000,B 90.000,C 0.000} C_DIS
LIN {X 44.617,Y -46.131,Z -163.782,A -90.000,B 90.000,C 0.000} C_DIS
LIN {X 44.861,Y -46.157,Z -163.521,A -90.000,B 90.000,C 0.000} C_DIS
LIN {X 45.017,Y -46.175,Z -163.364,A -90.000,B 90.000,C 0.000} C_DIS
LIN {X 45.262,Y -46.205,Z -163.134,A -90.000,B 90.000,C 0.000} C_DIS
LIN {X 45.418,Y -46.225,Z -162.996,A -90.000,B 90.000,C 0.000} C_DIS
LIN {X 45.589,Y -46.242,Z -162.850,A -90.000,B 90.000,C 0.000} C_DIS
LIN {X 45.945,Y -46.278,Z -162.558,A -90.000,B 90.000,C 0.000} C_DIS
LIN {X 46.057,Y -46.290,Z -162.473,A -90.000,B 90.000,C 0.000} C_DIS
LIN {X 46.232,Y -46.309,Z -162.346,A -90.000,B 90.000,C 0.000} C_DIS
LIN {X 46.590,Y -46.350,Z -162.094,A -90.000,B 90.000,C 0.000} C_DIS
LIN {X 46.799,Y -46.375,Z -161.956,A -90.000,B 90.000,C 0.000} C_DIS
LIN {X 47.178,Y -46.423,Z -161.725,A -90.000,B 90.000,C 0.000} C_DIS
LIN {X 47.412,Y -46.453,Z -161.592,A -90.000,B 90.000,C 0.000} C_DIS
LIN {X 47.725,Y -46.495,Z -161.428,A -90.000,B 90.000,C 0.000} C_DIS
LIN {X 47.822,Y -46.509,Z -161.380,A -90.000,B 90.000,C 0.000} C_DIS
LIN {X 48.239,Y -46.568,Z -161.189,A -90.000,B 90.000,C 0.000} C_DIS
LIN {X 48.533,Y -46.608,Z -161.066,A -90.000,B 90.000,C 0.000} C_DIS
LIN {X 48.737,Y -46.633,Z -160.988,A -90.000,B 90.000,C 0.000} C_DIS
LIN {X 49.043,Y -46.669,Z -160.882,A -90.000,B 90.000,C 0.000} C_DIS
LIN {X 49.275,Y -46.693,Z -160.810,A -90.000,B 90.000,C 0.000} C_DIS
LIN {X 49.583,Y -46.725,Z -160.724,A -90.000,B 90.000,C 0.000} C_DIS
LIN {X 49.878,Y -46.755,Z -160.650,A -90.000,B 90.000,C 0.000} C_DIS
LIN {X 50.174,Y -46.785,Z -160.588,A -90.000,B 90.000,C 0.000} C_DIS
LIN {X 50.476,Y -46.818,Z -160.537,A -90.000,B 90.000,C 0.000} C_DIS
LIN {X 50.553,Y -46.826,Z -160.526,A -90.000,B 90.000,C 0.000} C_DIS
LIN {X 51.163,Y -46.894,Z -160.444,A -90.000,B 90.000,C 0.000} C_DIS
LIN {X 51.487,Y -46.931,Z -160.414,A -90.000,B 90.000,C 0.000} C_DIS
LIN {X 51.679,Y -46.953,Z -160.402,A -90.000,B 90.000,C 0.000} C_DIS
LIN {X 51.734,Y -46.960,Z -160.401,A -90.000,B 90.000,C 0.000} C_DIS
LIN {X 52.027,Y -46.977,Z -160.394,A -90.000,B 90.000,C 0.000} C_DIS
LIN {X 52.272,Y -46.992,Z -160.396,A -90.000,B 90.000,C 0.000} C_DIS
LIN {X 52.615,Y -47.007,Z -160.408,A -90.000,B 90.000,C 0.000} C_DIS
LIN {X 52.897,Y -47.020,Z -160.428,A -90.000,B 90.000,C 0.000} C_DIS
LIN {X 53.131,Y -47.031,Z -160.451,A -90.000,B 90.000,C 0.000} C_DIS
LIN {X 53.355,Y -47.042,Z -160.475,A -90.000,B 90.000,C 0.000} C_DIS
LIN {X 53.774,Y -47.064,Z -160.539,A -90.000,B 90.000,C 0.000} C_DIS
LIN {X 54.046,Y -47.082,Z -160.589,A -90.000,B 90.000,C 0.000} C_DIS
LIN {X 54.370,Y -47.103,Z -160.660,A -90.000,B 90.000,C 0.000} C_DIS
LIN {X 54.839,Y -47.135,Z -160.783,A -90.000,B 90.000,C 0.000} C_DIS
LIN {X 54.949,Y -47.140,Z -160.816,A -90.000,B 90.000,C 0.000} C_DIS
LIN {X 55.141,Y -47.139,Z -160.875,A -90.000,B 90.000,C 0.000} C_DIS
LIN {X 55.393,Y -47.134,Z -160.960,A -90.000,B 90.000,C 0.000} C_DIS
LIN {X 55.701,Y -47.128,Z -161.077,A -90.000,B 90.000,C 0.000} C_DIS
LIN {X 55.986,Y -47.122,Z -161.191,A -90.000,B 90.000,C 0.000} C_DIS
LIN {X 56.148,Y -47.119,Z -161.263,A -90.000,B 90.000,C 0.000} C_DIS
LIN {X 56.422,Y -47.114,Z -161.392,A -90.000,B 90.000,C 0.000} C_DIS
LIN {X 56.734,Y -47.108,Z -161.549,A -90.000,B 90.000,C 0.000} C_DIS
LIN {X 56.912,Y -47.105,Z -161.645,A -90.000,B 90.000,C 0.000} C_DIS
LIN {X 57.247,Y -47.103,Z -161.842,A -90.000,B 90.000,C 0.000} C_DIS
LIN {X 57.523,Y -47.101,Z -162.014,A -90.000,B 90.000,C 0.000} C_DIS
LIN {X 57.769,Y -47.099,Z -162.179,A -90.000,B 90.000,C 0.000} C_DIS
LIN {X 58.038,Y -47.075,Z -162.373,A -90.000,B 90.000,C 0.000} C_DIS
LIN {X 58.303,Y -47.050,Z -162.579,A -90.000,B 90.000,C 0.000} C_DIS
LIN {X 58.565,Y -47.024,Z -162.797,A -90.000,B 90.000,C 0.000} C_DIS
LIN {X 58.798,Y -47.000,Z -163.005,A -90.000,B 90.000,C 0.000} C_DIS
LIN {X 59.055,Y -46.975,Z -163.249,A -90.000,B 90.000,C 0.000} C_DIS
LIN {X 59.210,Y -46.958,Z -163.404,A -90.000,B 90.000,C 0.000} C_DIS
LIN {X 59.518,Y -46.921,Z -163.737,A -90.000,B 90.000,C 0.000} C_DIS
LIN {X 59.772,Y -46.890,Z -164.034,A -90.000,B 90.000,C 0.000} C_DIS
LIN {X 59.837,Y -46.882,Z -164.114,A -90.000,B 90.000,C 0.000} C_DIS
LIN {X 60.090,Y -46.850,Z -164.444,A -90.000,B 90.000,C 0.000} C_DIS
LIN {X 60.289,Y -46.824,Z -164.728,A -90.000,B 90.000,C 0.000} C_DIS
LIN {X 60.406,Y -46.809,Z -164.901,A -90.000,B 90.000,C 0.000} C_DIS
LIN {X 60.470,Y -46.800,Z -164.999,A -90.000,B 90.000,C 0.000} C_DIS
LIN {X 60.599,Y -46.783,Z -165.211,A -90.000,B 90.000,C 0.000} C_DIS
LIN {X 60.709,Y -46.756,Z -165.400,A -90.000,B 90.000,C 0.000} C_DIS
LIN {X 60.784,Y -46.737,Z -165.535,A -90.000,B 90.000,C 0.000} C_DIS
LIN {X 60.937,Y -46.699,Z -165.826,A -90.000,B 90.000,C 0.000} C_DIS
LIN {X 61.027,Y -46.676,Z -166.011,A -90.000,B 90.000,C 0.000} C_DIS
LIN {X 61.127,Y -46.649,Z -166.229,A -90.000,B 90.000,C 0.000} C_DIS
LIN {X 61.256,Y -46.614,Z -166.526,A -90.000,B 90.000,C 0.000} C_DIS
LIN {X 61.323,Y -46.595,Z -166.695,A -90.000,B 90.000,C 0.000} C_DIS
LIN {X 61.480,Y -46.550,Z -167.125,A -90.000,B 90.000,C 0.000} C_DIS
LIN {X 61.608,Y -46.510,Z -167.515,A -90.000,B 90.000,C 0.000} C_DIS
LIN {X 61.699,Y -46.478,Z -167.821,A -90.000,B 90.000,C 0.000} C_DIS
LIN {X 61.742,Y -46.461,Z -167.985,A -90.000,B 90.000,C 0.000} C_DIS
LIN {X 61.811,Y -46.434,Z -168.252,A -90.000,B 90.000,C 0.000} C_DIS
LIN {X 61.870,Y -46.409,Z -168.516,A -90.000,B 90.000,C 0.000} C_DIS
LIN {X 61.902,Y -46.394,Z -168.682,A -90.000,B 90.000,C 0.000} C_DIS
LIN {X 61.940,Y -46.375,Z -168.904,A -90.000,B 90.000,C 0.000} C_DIS
LIN {X 61.971,Y -46.357,Z -169.132,A -90.000,B 90.000,C 0.000} C_DIS
LIN {X 61.998,Y -46.339,Z -169.354,A -90.000,B 90.000,C 0.000} C_DIS
LIN {X 62.059,Y -46.287,Z -170.069,A -90.000,B 90.000,C 0.000} C_DIS
LIN {X 62.071,Y -46.267,Z -170.368,A -90.000,B 90.000,C 0.000} C_DIS
LIN {X 62.074,Y -46.243,Z -170.772,A -90.000,B 90.000,C 0.000} C_DIS
LIN {X 62.067,Y -46.228,Z -171.074,A -90.000,B 90.000,C 0.000} C_DIS
LIN {X 62.054,Y -46.219,Z -171.284,A -90.000,B 90.000,C 0.000} C_DIS
LIN {X 62.028,Y -46.206,Z -171.594,A -90.000,B 90.000,C 0.000} C_DIS
LIN {X 61.920,Y -46.167,Z -172.633,A -90.000,B 90.000,C 0.000} C_DIS
LIN {X 61.903,Y -46.091,Z -173.999,A -90.000,B 90.000,C 0.000} C_DIS
LIN {X 61.901,Y -46.085,Z -174.145,A -90.000,B 90.000,C 0.000} C_DIS
LIN {X 62.162,Y -45.966,Z -175.474,A -90.000,B 90.000,C 0.000} C_DIS
LIN {X 62.234,Y -45.938,Z -175.746,A -90.000,B 90.000,C 0.000} C_DIS
LIN {X 62.292,Y -45.913,Z -175.996,A -90.000,B 90.000,C 0.000} C_DIS
LIN {X 62.354,Y -45.885,Z -176.318,A -90.000,B 90.000,C 0.000} C_DIS
LIN {X 62.424,Y -45.851,Z -176.725,A -90.000,B 90.000,C 0.000} C_DIS
LIN {X 62.461,Y -45.831,Z -176.975,A -90.000,B 90.000,C 0.000} C_DIS
LIN {X 62.494,Y -45.818,Z -177.240,A -90.000,B 90.000,C 0.000} C_DIS
LIN {X 62.601,Y -45.766,Z -178.498,A -90.000,B 90.000,C 0.000} C_DIS
LIN {X 62.619,Y -45.755,Z -178.770,A -90.000,B 90.000,C 0.000} C_DIS
LIN {X 62.627,Y -45.750,Z -178.914,A -90.000,B 90.000,C 0.000} C_DIS
LIN {X 62.642,Y -45.732,Z -179.471,A -90.000,B 90.000,C 0.000} C_DIS
LIN {X 62.675,Y -45.718,Z -179.701,A -90.000,B 90.000,C 0.000} C_DIS
LIN {X 62.699,Y -45.712,Z -179.875,A -90.000,B 90.000,C 0.000} C_DIS
LIN {X 62.860,Y -45.669,Z -181.286,A -90.000,B 90.000,C 0.000} C_DIS
LIN {X 63.094,Y -45.612,Z -182.241,A -90.000,B 90.000,C 0.000} C_DIS
LIN {X 63.387,Y -45.509,Z -183.464,A -90.000,B 90.000,C 0.000} C_DIS
LIN {X 63.431,Y -45.493,Z -183.673,A -90.000,B 90.000,C 0.000} C_DIS
LIN {X 63.503,Y -45.466,Z -184.072,A -90.000,B 90.000,C 0.000} C_DIS
LIN {X 63.540,Y -45.453,Z -184.301,A -90.000,B 90.000,C 0.000} C_DIS
LIN {X 63.584,Y -45.434,Z -184.639,A -90.000,B 90.000,C 0.000} C_DIS
LIN {X 63.613,Y -45.422,Z -184.919,A -90.000,B 90.000,C 0.000} C_DIS
LIN {X 63.641,Y -45.408,Z -185.258,A -90.000,B 90.000,C 0.000} C_DIS
LIN {X 63.658,Y -45.398,Z -185.573,A -90.000,B 90.000,C 0.000} C_DIS
LIN {X 63.709,Y -45.341,Z -187.899,A -90.000,B 90.000,C 0.000} C_DIS
LIN {X 63.719,Y -45.322,Z -188.484,A -90.000,B 90.000,C 0.000} C_DIS
LIN {X 63.725,Y -45.308,Z -188.920,A -90.000,B 90.000,C 0.000} C_DIS
LIN {X 63.725,Y -60.000,Z -188.920,A -90.000,B 90.000,C 0.000} C_DIS
LIN {X 41.812,Y -60.000,Z -163.444,A -90.000,B 90.000,C 0.000} C_DIS
LIN {X 41.812,Y -45.308,Z -163.444,A -90.000,B 90.000,C 0.000} C_DIS
LIN {X 42.851,Y -45.528,Z -162.750,A -90.000,B 90.000,C 0.000} C_DIS
LIN {X 42.907,Y -45.537,Z -162.714,A -90.000,B 90.000,C 0.000} C_DIS
LIN {X 43.135,Y -45.574,Z -162.555,A -90.000,B 90.000,C 0.000} C_DIS
LIN {X 43.239,Y -45.584,Z -162.439,A -90.000,B 90.000,C 0.000} C_DIS
LIN {X 43.529,Y -45.615,Z -162.131,A -90.000,B 90.000,C 0.000} C_DIS
LIN {X 43.731,Y -45.638,Z -161.929,A -90.000,B 90.000,C 0.000} C_DIS
LIN {X 44.028,Y -45.675,Z -161.651,A -90.000,B 90.000,C 0.000} C_DIS
LIN {X 44.395,Y -45.725,Z -161.331,A -90.000,B 90.000,C 0.000} C_DIS
LIN {X 44.818,Y -45.785,Z -160.981,A -90.000,B 90.000,C 0.000} C_DIS
LIN {X 44.953,Y -45.805,Z -160.877,A -90.000,B 90.000,C 0.000} C_DIS
LIN {X 45.200,Y -45.844,Z -160.696,A -90.000,B 90.000,C 0.000} C_DIS
LIN {X 45.473,Y -45.888,Z -160.500,A -90.000,B 90.000,C 0.000} C_DIS
LIN {X 45.612,Y -45.911,Z -160.404,A -90.000,B 90.000,C 0.000} C_DIS
LIN {X 45.821,Y -45.946,Z -160.265,A -90.000,B 90.000,C 0.000} C_DIS
LIN {X 46.252,Y -46.018,Z -159.999,A -90.000,B 90.000,C 0.000} C_DIS
LIN {X 46.542,Y -46.067,Z -159.833,A -90.000,B 90.000,C 0.000} C_DIS
LIN {X 46.903,Y -46.118,Z -159.644,A -90.000,B 90.000,C 0.000} C_DIS
LIN {X 47.067,Y -46.142,Z -159.565,A -90.000,B 90.000,C 0.000} C_DIS
LIN {X 47.521,Y -46.210,Z -159.357,A -90.000,B 90.000,C 0.000} C_DIS
LIN {X 47.864,Y -46.263,Z -159.214,A -90.000,B 90.000,C 0.000} C_DIS
LIN {X 48.132,Y -46.304,Z -159.111,A -90.000,B 90.000,C 0.000} C_DIS
LIN {X 48.500,Y -46.362,Z -158.982,A -90.000,B 90.000,C 0.000} C_DIS
LIN {X 48.766,Y -46.404,Z -158.898,A -90.000,B 90.000,C 0.000} C_DIS
LIN {X 49.130,Y -46.464,Z -158.793,A -90.000,B 90.000,C 0.000} C_DIS
LIN {X 49.232,Y -46.481,Z -158.767,A -90.000,B 90.000,C 0.000} C_DIS
LIN {X 49.402,Y -46.503,Z -158.724,A -90.000,B 90.000,C 0.000} C_DIS
LIN {X 49.634,Y -46.535,Z -158.672,A -90.000,B 90.000,C 0.000} C_DIS
LIN {X 49.771,Y -46.553,Z -158.643,A -90.000,B 90.000,C 0.000} C_DIS
LIN {X 49.895,Y -46.567,Z -158.620,A -90.000,B 90.000,C 0.000} C_DIS
LIN {X 50.252,Y -46.609,Z -158.560,A -90.000,B 90.000,C 0.000} C_DIS
LIN {X 50.926,Y -46.690,Z -158.468,A -90.000,B 90.000,C 0.000} C_DIS
LIN {X 51.012,Y -46.701,Z -158.459,A -90.000,B 90.000,C 0.000} C_DIS
LIN {X 51.329,Y -46.740,Z -158.430,A -90.000,B 90.000,C 0.000} C_DIS
LIN {X 51.639,Y -46.780,Z -158.410,A -90.000,B 90.000,C 0.000} C_DIS
LIN {X 52.048,Y -46.833,Z -158.399,A -90.000,B 90.000,C 0.000} C_DIS
LIN {X 52.350,Y -46.873,Z -158.401,A -90.000,B 90.000,C 0.000} C_DIS
LIN {X 52.400,Y -46.879,Z -158.402,A -90.000,B 90.000,C 0.000} C_DIS
LIN {X 52.761,Y -46.902,Z -158.416,A -90.000,B 90.000,C 0.000} C_DIS
LIN {X 53.042,Y -46.918,Z -158.436,A -90.000,B 90.000,C 0.000} C_DIS
LIN {X 53.328,Y -46.935,Z -158.463,A -90.000,B 90.000,C 0.000} C_DIS
LIN {X 53.578,Y -46.950,Z -158.490,A -90.000,B 90.000,C 0.000} C_DIS
LIN {X 54.038,Y -46.978,Z -158.558,A -90.000,B 90.000,C 0.000} C_DIS
LIN {X 54.159,Y -46.986,Z -158.578,A -90.000,B 90.000,C 0.000} C_DIS
LIN {X 54.479,Y -47.006,Z -158.638,A -90.000,B 90.000,C 0.000} C_DIS
LIN {X 54.803,Y -47.028,Z -158.710,A -90.000,B 90.000,C 0.000} C_DIS
LIN {X 55.115,Y -47.050,Z -158.789,A -90.000,B 90.000,C 0.000} C_DIS
LIN {X 55.409,Y -47.070,Z -158.867,A -90.000,B 90.000,C 0.000} C_DIS
LIN {X 55.574,Y -47.080,Z -158.916,A -90.000,B 90.000,C 0.000} C_DIS
LIN {X 55.734,Y -47.080,Z -158.966,A -90.000,B 90.000,C 0.000} C_DIS
LIN {X 56.098,Y -47.076,Z -159.090,A -90.000,B 90.000,C 0.000} C_DIS
LIN {X 56.432,Y -47.072,Z -159.216,A -90.000,B 90.000,C 0.000} C_DIS
LIN {X 56.793,Y -47.068,Z -159.362,A -90.000,B 90.000,C 0.000} C_DIS
LIN {X 56.998,Y -47.066,Z -159.453,A -90.000,B 90.000,C 0.000} C_DIS
LIN {X 57.320,Y -47.063,Z -159.605,A -90.000,B 90.000,C 0.000} C_DIS
LIN {X 57.688,Y -47.060,Z -159.791,A -90.000,B 90.000,C 0.000} C_DIS
LIN {X 57.940,Y -47.058,Z -159.930,A -90.000,B 90.000,C 0.000} C_DIS
LIN {X 58.301,Y -47.056,Z -160.144,A -90.000,B 90.000,C 0.000} C_DIS
LIN {X 58.393,Y -47.054,Z -160.201,A -90.000,B 90.000,C 0.000} C_DIS
LIN {X 58.635,Y -47.033,Z -160.353,A -90.000,B 90.000,C 0.000} C_DIS
LIN {X 58.935,Y -47.005,Z -160.556,A -90.000,B 90.000,C 0.000} C_DIS
LIN {X 58.984,Y -47.000,Z -160.592,A -90.000,B 90.000,C 0.000} C_DIS
LIN {X 59.257,Y -46.973,Z -160.791,A -90.000,B 90.000,C 0.000} C_DIS
LIN {X 59.572,Y -46.942,Z -161.037,A -90.000,B 90.000,C 0.000} C_DIS
LIN {X 59.890,Y -46.910,Z -161.303,A -90.000,B 90.000,C 0.000} C_DIS
LIN {X 60.163,Y -46.884,Z -161.549,A -90.000,B 90.000,C 0.000} C_DIS
LIN {X 60.464,Y -46.856,Z -161.834,A -90.000,B 90.000,C 0.000} C_DIS
LIN {X 60.669,Y -46.836,Z -162.042,A -90.000,B 90.000,C 0.000} C_DIS
LIN {X 61.026,Y -46.801,Z -162.429,A -90.000,B 90.000,C 0.000} C_DIS
LIN {X 61.328,Y -46.772,Z -162.782,A -90.000,B 90.000,C 0.000} C_DIS
LIN {X 61.414,Y -46.756,Z -162.891,A -90.000,B 90.000,C 0.000} C_DIS
LIN {X 61.665,Y -46.706,Z -163.220,A -90.000,B 90.000,C 0.000} C_DIS
LIN {X 61.715,Y -46.696,Z -163.288,A -90.000,B 90.000,C 0.000} C_DIS
LIN {X 61.948,Y -46.649,Z -163.624,A -90.000,B 90.000,C 0.000} C_DIS
LIN {X 62.077,Y -46.623,Z -163.817,A -90.000,B 90.000,C 0.000} C_DIS
LIN {X 62.163,Y -46.605,Z -163.953,A -90.000,B 90.000,C 0.000} C_DIS
LIN {X 62.398,Y -46.549,Z -164.349,A -90.000,B 90.000,C 0.000} C_DIS
LIN {X 62.534,Y -46.516,Z -164.592,A -90.000,B 90.000,C 0.000} C_DIS
LIN {X 62.711,Y -46.471,Z -164.931,A -90.000,B 90.000,C 0.000} C_DIS
LIN {X 62.819,Y -46.443,Z -165.155,A -90.000,B 90.000,C 0.000} C_DIS
LIN {X 62.946,Y -46.409,Z -165.432,A -90.000,B 90.000,C 0.000} C_DIS
LIN {X 63.091,Y -46.369,Z -165.768,A -90.000,B 90.000,C 0.000} C_DIS
LIN {X 63.179,Y -46.344,Z -165.991,A -90.000,B 90.000,C 0.000} C_DIS
LIN {X 63.357,Y -46.291,Z -166.484,A -90.000,B 90.000,C 0.000} C_DIS
LIN {X 63.496,Y -46.247,Z -166.911,A -90.000,B 90.000,C 0.000} C_DIS
LIN {X 63.542,Y -46.232,Z -167.063,A -90.000,B 90.000,C 0.000} C_DIS
LIN {X 63.608,Y -46.206,Z -167.291,A -90.000,B 90.000,C 0.000} C_DIS
LIN {X 63.737,Y -46.152,Z -167.794,A -90.000,B 90.000,C 0.000} C_DIS
LIN {X 63.774,Y -46.134,Z -167.963,A -90.000,B 90.000,C 0.000} C_DIS
LIN {X 63.795,Y -46.123,Z -168.058,A -90.000,B 90.000,C 0.000} C_DIS
LIN {X 63.847,Y -46.091,Z -168.323,A -90.000,B 90.000,C 0.000} C_DIS
LIN {X 63.894,Y -46.058,Z -168.616,A -90.000,B 90.000,C 0.000} C_DIS
LIN {X 63.941,Y -46.020,Z -168.986,A -90.000,B 90.000,C 0.000} C_DIS
LIN {X 63.960,Y -46.002,Z -169.162,A -90.000,B 90.000,C 0.000} C_DIS
LIN {X 64.018,Y -45.935,Z -169.877,A -90.000,B 90.000,C 0.000} C_DIS
LIN {X 64.023,Y -45.927,Z -169.964,A -90.000,B 90.000,C 0.000} C_DIS
LIN {X 64.036,Y -45.896,Z -170.332,A -90.000,B 90.000,C 0.000} C_DIS
LIN {X 64.037,Y -45.859,Z -170.808,A -90.000,B 90.000,C 0.000} C_DIS
LIN {X 64.025,Y -45.833,Z -171.173,A -90.000,B 90.000,C 0.000} C_DIS
LIN {X 64.013,Y -45.821,Z -171.357,A -90.000,B 90.000,C 0.000} C_DIS
LIN {X 63.977,Y -45.799,Z -171.782,A -90.000,B 90.000,C 0.000} C_DIS
LIN {X 63.876,Y -45.754,Z -172.724,A -90.000,B 90.000,C 0.000} C_DIS
LIN {X 63.858,Y -45.673,Z -173.939,A -90.000,B 90.000,C 0.000} C_DIS
LIN {X 63.937,Y -45.628,Z -174.347,A -90.000,B 90.000,C 0.000} C_DIS
LIN {X 64.064,Y -45.570,Z -174.996,A -90.000,B 90.000,C 0.000} C_DIS
LIN {X 64.137,Y -45.542,Z -175.275,A -90.000,B 90.000,C 0.000} C_DIS
LIN {X 64.194,Y -45.518,Z -175.521,A -90.000,B 90.000,C 0.000} C_DIS
LIN {X 64.271,Y -45.484,Z -175.912,A -90.000,B 90.000,C 0.000} C_DIS
LIN {X 64.356,Y -45.443,Z -176.406,A -90.000,B 90.000,C 0.000} C_DIS
LIN {X 64.401,Y -45.420,Z -176.715,A -90.000,B 90.000,C 0.000} C_DIS
LIN {X 64.440,Y -45.395,Z -177.057,A -90.000,B 90.000,C 0.000} C_DIS
LIN {X 64.461,Y -45.379,Z -177.313,A -90.000,B 90.000,C 0.000} C_DIS
LIN {X 64.513,Y -45.354,Z -177.931,A -90.000,B 90.000,C 0.000} C_DIS
LIN {X 64.547,Y -45.328,Z -178.352,A -90.000,B 90.000,C 0.000} C_DIS
LIN {X 64.567,Y -45.308,Z -178.689,A -90.000,B 90.000,C 0.000} C_DIS
LIN {X 64.567,Y -60.000,Z -178.689,A -90.000,B 90.000,C 0.000} C_DIS
LIN {X 44.233,Y -60.000,Z -159.025,A -90.000,B 90.000,C 0.000} C_DIS
LIN {X 44.233,Y -45.308,Z -159.025,A -90.000,B 90.000,C 0.000} C_DIS
LIN {X 44.491,Y -45.351,Z -158.842,A -90.000,B 90.000,C 0.000} C_DIS
LIN {X 44.638,Y -45.376,Z -158.741,A -90.000,B 90.000,C 0.000} C_DIS
LIN {X 44.871,Y -45.417,Z -158.586,A -90.000,B 90.000,C 0.000} C_DIS
LIN {X 45.358,Y -45.506,Z -158.284,A -90.000,B 90.000,C 0.000} C_DIS
LIN {X 45.646,Y -45.561,Z -158.118,A -90.000,B 90.000,C 0.000} C_DIS
LIN {X 46.113,Y -45.652,Z -157.867,A -90.000,B 90.000,C 0.000} C_DIS
LIN {X 46.313,Y -45.693,Z -157.767,A -90.000,B 90.000,C 0.000} C_DIS
LIN {X 46.836,Y -45.799,Z -157.524,A -90.000,B 90.000,C 0.000} C_DIS
LIN {X 47.212,Y -45.871,Z -157.364,A -90.000,B 90.000,C 0.000} C_DIS
LIN {X 47.461,Y -45.920,Z -157.266,A -90.000,B 90.000,C 0.000} C_DIS
LIN {X 47.526,Y -45.930,Z -157.242,A -90.000,B 90.000,C 0.000} C_DIS
LIN {X 47.959,Y -46.000,Z -157.091,A -90.000,B 90.000,C 0.000} C_DIS
LIN {X 48.274,Y -46.052,Z -156.992,A -90.000,B 90.000,C 0.000} C_DIS
LIN {X 48.693,Y -46.124,Z -156.871,A -90.000,B 90.000,C 0.000} C_DIS
LIN {X 49.014,Y -46.180,Z -156.789,A -90.000,B 90.000,C 0.000} C_DIS
LIN {X 49.362,Y -46.242,Z -156.710,A -90.000,B 90.000,C 0.000} C_DIS
LIN {X 49.602,Y -46.286,Z -156.661,A -90.000,B 90.000,C 0.000} C_DIS
LIN {X 50.013,Y -46.362,Z -156.590,A -90.000,B 90.000,C 0.000} C_DIS
LIN {X 50.686,Y -46.451,Z -156.497,A -90.000,B 90.000,C 0.000} C_DIS
LIN {X 50.870,Y -46.474,Z -156.477,A -90.000,B 90.000,C 0.000} C_DIS
LIN {X 51.232,Y -46.521,Z -156.444,A -90.000,B 90.000,C 0.000} C_DIS
LIN {X 51.613,Y -46.571,Z -156.421,A -90.000,B 90.000,C 0.000} C_DIS
LIN {X 52.076,Y -46.633,Z -156.410,A -90.000,B 90.000,C 0.000} C_DIS
LIN {X 52.454,Y -46.683,Z -156.413,A -90.000,B 90.000,C 0.000} C_DIS
LIN {X 52.922,Y -46.746,Z -156.429,A -90.000,B 90.000,C 0.000} C_DIS
LIN {X 53.102,Y -46.771,Z -156.440,A -90.000,B 90.000,C 0.000} C_DIS
LIN {X 53.180,Y -46.779,Z -156.445,A -90.000,B 90.000,C 0.000} C_DIS
LIN {X 53.583,Y -46.802,Z -156.483,A -90.000,B 90.000,C 0.000} C_DIS
LIN {X 53.880,Y -46.820,Z -156.517,A -90.000,B 90.000,C 0.000} C_DIS
LIN {X 53.922,Y -46.822,Z -156.523,A -90.000,B 90.000,C 0.000} C_DIS
LIN {X 54.461,Y -46.856,Z -156.605,A -90.000,B 90.000,C 0.000} C_DIS
LIN {X 54.600,Y -46.866,Z -156.630,A -90.000,B 90.000,C 0.000} C_DIS
LIN {X 54.918,Y -46.889,Z -156.690,A -90.000,B 90.000,C 0.000} C_DIS
LIN {X 55.307,Y -46.919,Z -156.777,A -90.000,B 90.000,C 0.000} C_DIS
LIN {X 55.776,Y -46.955,Z -156.898,A -90.000,B 90.000,C 0.000} C_DIS
LIN {X 55.985,Y -46.970,Z -156.955,A -90.000,B 90.000,C 0.000} C_DIS
LIN {X 56.194,Y -46.984,Z -157.017,A -90.000,B 90.000,C 0.000} C_DIS
LIN {X 56.315,Y -46.986,Z -157.055,A -90.000,B 90.000,C 0.000} C_DIS
LIN {X 56.804,Y -46.983,Z -157.221,A -90.000,B 90.000,C 0.000} C_DIS
LIN {X 57.181,Y -46.980,Z -157.364,A -90.000,B 90.000,C 0.000} C_DIS
LIN {X 57.604,Y -46.978,Z -157.536,A -90.000,B 90.000,C 0.000} C_DIS
LIN {X 57.855,Y -46.979,Z -157.649,A -90.000,B 90.000,C 0.000} C_DIS
LIN {X 58.222,Y -46.980,Z -157.822,A -90.000,B 90.000,C 0.000} C_DIS
LIN {X 58.651,Y -46.983,Z -158.040,A -90.000,B 90.000,C 0.000} C_DIS
LIN {X 58.960,Y -46.984,Z -158.212,A -90.000,B 90.000,C 0.000} C_DIS
LIN {X 59.031,Y -46.981,Z -158.254,A -90.000,B 90.000,C 0.000} C_DIS
LIN {X 59.366,Y -46.957,Z -158.454,A -90.000,B 90.000,C 0.000} C_DIS
LIN {X 59.693,Y -46.931,Z -158.659,A -90.000,B 90.000,C 0.000} C_DIS
LIN {X 60.099,Y -46.899,Z -158.934,A -90.000,B 90.000,C 0.000} C_DIS
LIN {X 60.480,Y -46.869,Z -159.212,A -90.000,B 90.000,C 0.000} C_DIS
LIN {X 60.847,Y -46.840,Z -159.500,A -90.000,B 90.000,C 0.000} C_DIS
LIN {X 61.218,Y -46.812,Z -159.810,A -90.000,B 90.000,C 0.000} C_DIS
LIN {X 61.483,Y -46.791,Z -160.049,A -90.000,B 90.000,C 0.000} C_DIS
LIN {X 61.674,Y -46.773,Z -160.228,A -90.000,B 90.000,C 0.000} C_DIS
LIN {X 61.881,Y -46.753,Z -160.426,A -90.000,B 90.000,C 0.000} C_DIS
LIN {X 62.024,Y -46.740,Z -160.571,A -90.000,B 90.000,C 0.000} C_DIS
LIN {X 62.132,Y -46.719,Z -160.683,A -90.000,B 90.000,C 0.000} C_DIS
LIN {X 62.535,Y -46.643,Z -161.126,A -90.000,B 90.000,C 0.000} C_DIS
LIN {X 62.876,Y -46.577,Z -161.530,A -90.000,B 90.000,C 0.000} C_DIS
LIN {X 62.981,Y -46.557,Z -161.664,A -90.000,B 90.000,C 0.000} C_DIS
LIN {X 63.258,Y -46.503,Z -162.028,A -90.000,B 90.000,C 0.000} C_DIS
LIN {X 63.366,Y -46.481,Z -162.179,A -90.000,B 90.000,C 0.000} C_DIS
LIN {X 63.583,Y -46.438,Z -162.492,A -90.000,B 90.000,C 0.000} C_DIS
LIN {X 63.746,Y -46.405,Z -162.736,A -90.000,B 90.000,C 0.000} C_DIS
LIN {X 63.886,Y -46.376,Z -162.963,A -90.000,B 90.000,C 0.000} C_DIS
LIN {X 64.119,Y -46.327,Z -163.354,A -90.000,B 90.000,C 0.000} C_DIS
LIN {X 64.286,Y -46.292,Z -163.652,A -90.000,B 90.000,C 0.000} C_DIS
LIN {X 64.466,Y -46.253,Z -163.998,A -90.000,B 90.000,C 0.000} C_DIS
LIN {X 64.614,Y -46.210,Z -164.305,A -90.000,B 90.000,C 0.000} C_DIS
LIN {X 64.771,Y -46.163,Z -164.652,A -90.000,B 90.000,C 0.000} C_DIS
LIN {X 64.925,Y -46.105,Z -165.017,A -90.000,B 90.000,C 0.000} C_DIS
LIN {X 65.030,Y -46.063,Z -165.290,A -90.000,B 90.000,C 0.000} C_DIS
LIN {X 65.226,Y -45.982,Z -165.842,A -90.000,B 90.000,C 0.000} C_DIS
LIN {X 65.377,Y -45.916,Z -166.316,A -90.000,B 90.000,C 0.000} C_DIS
LIN {X 65.507,Y -45.856,Z -166.769,A -90.000,B 90.000,C 0.000} C_DIS
LIN {X 65.648,Y -45.786,Z -167.331,A -90.000,B 90.000,C 0.000} C_DIS
LIN {X 65.716,Y -45.749,Z -167.643,A -90.000,B 90.000,C 0.000} C_DIS
LIN {X 65.778,Y -45.713,Z -167.967,A -90.000,B 90.000,C 0.000} C_DIS
LIN {X 65.834,Y -45.676,Z -168.318,A -90.000,B 90.000,C 0.000} C_DIS
LIN {X 65.886,Y -45.632,Z -168.733,A -90.000,B 90.000,C 0.000} C_DIS
LIN {X 65.911,Y -45.608,Z -168.966,A -90.000,B 90.000,C 0.000} C_DIS
LIN {X 65.960,Y -45.549,Z -169.570,A -90.000,B 90.000,C 0.000} C_DIS
LIN {X 65.977,Y -45.526,Z -169.811,A -90.000,B 90.000,C 0.000} C_DIS
LIN {X 65.993,Y -45.483,Z -170.299,A -90.000,B 90.000,C 0.000} C_DIS
LIN {X 65.992,Y -45.440,Z -170.841,A -90.000,B 90.000,C 0.000} C_DIS
LIN {X 65.981,Y -45.417,Z -171.163,A -90.000,B 90.000,C 0.000} C_DIS
LIN {X 65.975,Y -45.407,Z -171.302,A -90.000,B 90.000,C 0.000} C_DIS
LIN {X 65.959,Y -45.393,Z -171.529,A -90.000,B 90.000,C 0.000} C_DIS
LIN {X 65.921,Y -45.369,Z -171.969,A -90.000,B 90.000,C 0.000} C_DIS
LIN {X 65.831,Y -45.328,Z -172.819,A -90.000,B 90.000,C 0.000} C_DIS
LIN {X 65.826,Y -45.308,Z -173.106,A -90.000,B 90.000,C 0.000} C_DIS
LIN {X 65.826,Y -60.000,Z -173.106,A -90.000,B 90.000,C 0.000} C_DIS
LIN {X 46.248,Y -60.000,Z -155.674,A -90.000,B 90.000,C 0.000} C_DIS
LIN {X 46.248,Y -45.308,Z -155.674,A -90.000,B 90.000,C 0.000} C_DIS
LIN {X 46.586,Y -45.381,Z -155.529,A -90.000,B 90.000,C 0.000} C_DIS
LIN {X 46.955,Y -45.462,Z -155.383,A -90.000,B 90.000,C 0.000} C_DIS
LIN {X 47.450,Y -45.573,Z -155.204,A -90.000,B 90.000,C 0.000} C_DIS
LIN {X 47.796,Y -45.652,Z -155.091,A -90.000,B 90.000,C 0.000} C_DIS
LIN {X 48.267,Y -45.749,Z -154.953,A -90.000,B 90.000,C 0.000} C_DIS
LIN {X 48.349,Y -45.766,Z -154.932,A -90.000,B 90.000,C 0.000} C_DIS
LIN {X 48.642,Y -45.819,Z -154.857,A -90.000,B 90.000,C 0.000} C_DIS
LIN {X 49.270,Y -45.936,Z -154.720,A -90.000,B 90.000,C 0.000} C_DIS
LIN {X 49.770,Y -46.032,Z -154.632,A -90.000,B 90.000,C 0.000} C_DIS
LIN {X 50.501,Y -46.176,Z -154.525,A -90.000,B 90.000,C 0.000} C_DIS
LIN {X 50.799,Y -46.235,Z -154.491,A -90.000,B 90.000,C 0.000} C_DIS
LIN {X 51.065,Y -46.272,Z -154.467,A -90.000,B 90.000,C 0.000} C_DIS
LIN {X 51.446,Y -46.322,Z -154.442,A -90.000,B 90.000,C 0.000} C_DIS
LIN {X 51.593,Y -46.341,Z -154.435,A -90.000,B 90.000,C 0.000} C_DIS
LIN {X 52.122,Y -46.412,Z -154.422,A -90.000,B 90.000,C 0.000} C_DIS
LIN {X 52.551,Y -46.472,Z -154.426,A -90.000,B 90.000,C 0.000} C_DIS
LIN {X 53.076,Y -46.546,Z -154.445,A -90.000,B 90.000,C 0.000} C_DIS
LIN {X 53.377,Y -46.590,Z -154.464,A -90.000,B 90.000,C 0.000} C_DIS
LIN {X 53.808,Y -46.654,Z -154.501,A -90.000,B 90.000,C 0.000} C_DIS
LIN {X 53.882,Y -46.665,Z -154.509,A -90.000,B 90.000,C 0.000} C_DIS
LIN {X 54.182,Y -46.685,Z -154.545,A -90.000,B 90.000,C 0.000} C_DIS
LIN {X 54.818,Y -46.730,Z -154.641,A -90.000,B 90.000,C 0.000} C_DIS
LIN {X 54.983,Y -46.742,Z -154.671,A -90.000,B 90.000,C 0.000} C_DIS
LIN {X 55.355,Y -46.770,Z -154.742,A -90.000,B 90.000,C 0.000} C_DIS
LIN {X 55.816,Y -46.806,Z -154.846,A -90.000,B 90.000,C 0.000} C_DIS
LIN {X 56.307,Y -46.846,Z -154.973,A -90.000,B 90.000,C 0.000} C_DIS
LIN {X 56.547,Y -46.866,Z -155.038,A -90.000,B 90.000,C 0.000} C_DIS
LIN {X 56.908,Y -46.883,Z -155.147,A -90.000,B 90.000,C 0.000} C_DIS
LIN {X 57.445,Y -46.886,Z -155.329,A -90.000,B 90.000,C 0.000} C_DIS
LIN {X 57.935,Y -46.889,Z -155.514,A -90.000,B 90.000,C 0.000} C_DIS
LIN {X 58.419,Y -46.893,Z -155.712,A -90.000,B 90.000,C 0.000} C_DIS
LIN {X 58.655,Y -46.896,Z -155.817,A -90.000,B 90.000,C 0.000} C_DIS
LIN {X 59.128,Y -46.898,Z -156.041,A -90.000,B 90.000,C 0.000} C_DIS
LIN {X 59.607,Y -46.900,Z -156.285,A -90.000,B 90.000,C 0.000} C_DIS
LIN {X 59.696,Y -46.895,Z -156.335,A -90.000,B 90.000,C 0.000} C_DIS
LIN {X 60.012,Y -46.871,Z -156.514,A -90.000,B 90.000,C 0.000} C_DIS
LIN {X 60.421,Y -46.839,Z -156.759,A -90.000,B 90.000,C 0.000} C_DIS
LIN {X 60.805,Y -46.810,Z -157.001,A -90.000,B 90.000,C 0.000} C_DIS
LIN {X 61.270,Y -46.775,Z -157.317,A -90.000,B 90.000,C 0.000} C_DIS
LIN {X 61.705,Y -46.743,Z -157.636,A -90.000,B 90.000,C 0.000} C_DIS
LIN {X 62.126,Y -46.712,Z -157.967,A -90.000,B 90.000,C 0.000} C_DIS
LIN {X 62.545,Y -46.680,Z -158.320,A -90.000,B 90.000,C 0.000} C_DIS
LIN {X 62.675,Y -46.671,Z -158.437,A -90.000,B 90.000,C 0.000} C_DIS
LIN {X 62.809,Y -46.649,Z -158.558,A -90.000,B 90.000,C 0.000} C_DIS
LIN {X 63.147,Y -46.595,Z -158.879,A -90.000,B 90.000,C 0.000} C_DIS
LIN {X 63.249,Y -46.578,Z -158.978,A -90.000,B 90.000,C 0.000} C_DIS
LIN {X 63.548,Y -46.530,Z -159.283,A -90.000,B 90.000,C 0.000} C_DIS
LIN {X 64.010,Y -46.455,Z -159.789,A -90.000,B 90.000,C 0.000} C_DIS
LIN {X 64.426,Y -46.388,Z -160.281,A -90.000,B 90.000,C 0.000} C_DIS
LIN {X 64.564,Y -46.365,Z -160.457,A -90.000,B 90.000,C 0.000} C_DIS
LIN {X 64.808,Y -46.323,Z -160.777,A -90.000,B 90.000,C 0.000} C_DIS
LIN {X 64.857,Y -46.314,Z -160.842,A -90.000,B 90.000,C 0.000} C_DIS
LIN {X 64.989,Y -46.288,Z -161.026,A -90.000,B 90.000,C 0.000} C_DIS
LIN {X 65.212,Y -46.243,Z -161.347,A -90.000,B 90.000,C 0.000} C_DIS
LIN {X 65.311,Y -46.220,Z -161.496,A -90.000,B 90.000,C 0.000} C_DIS
LIN {X 65.422,Y -46.191,Z -161.667,A -90.000,B 90.000,C 0.000} C_DIS
LIN {X 65.585,Y -46.148,Z -161.932,A -90.000,B 90.000,C 0.000} C_DIS
LIN {X 65.837,Y -46.071,Z -162.363,A -90.000,B 90.000,C 0.000} C_DIS
LIN {X 66.028,Y -46.012,Z -162.711,A -90.000,B 90.000,C 0.000} C_DIS
LIN {X 66.242,Y -45.943,Z -163.132,A -90.000,B 90.000,C 0.000} C_DIS
LIN {X 66.397,Y -45.893,Z -163.456,A -90.000,B 90.000,C 0.000} C_DIS
LIN {X 66.571,Y -45.835,Z -163.845,A -90.000,B 90.000,C 0.000} C_DIS
LIN {X 66.749,Y -45.774,Z -164.264,A -90.000,B 90.000,C 0.000} C_DIS
LIN {X 66.888,Y -45.724,Z -164.630,A -90.000,B 90.000,C 0.000} C_DIS
LIN {X 67.027,Y -45.673,Z -165.018,A -90.000,B 90.000,C 0.000} C_DIS
LIN {X 67.090,Y -45.646,Z -165.201,A -90.000,B 90.000,C 0.000} C_DIS
LIN {X 67.255,Y -45.573,Z -165.721,A -90.000,B 90.000,C 0.000} C_DIS
LIN {X 67.406,Y -45.503,Z -166.249,A -90.000,B 90.000,C 0.000} C_DIS
LIN {X 67.560,Y -45.424,Z -166.871,A -90.000,B 90.000,C 0.000} C_DIS
LIN {X 67.639,Y -45.380,Z -167.234,A -90.000,B 90.000,C 0.000} C_DIS
LIN {X 67.688,Y -45.351,Z -167.495,A -90.000,B 90.000,C 0.000} C_DIS
LIN {X 67.718,Y -45.326,Z -167.666,A -90.000,B 90.000,C 0.000} C_DIS
LIN {X 67.738,Y -45.308,Z -167.798,A -90.000,B 90.000,C 0.000} C_DIS
LIN {X 67.738,Y -60.000,Z -167.798,A -90.000,B 90.000,C 0.000} C_DIS
LIN {X 47.936,Y -60.000,Z -153.029,A -90.000,B 90.000,C 0.000} C_DIS
LIN {X 47.936,Y -45.308,Z -153.029,A -90.000,B 90.000,C 0.000} C_DIS
LIN {X 48.293,Y -45.395,Z -152.934,A -90.000,B 90.000,C 0.000} C_DIS
LIN {X 48.697,Y -45.495,Z -152.841,A -90.000,B 90.000,C 0.000} C_DIS
LIN {X 49.002,Y -45.556,Z -152.775,A -90.000,B 90.000,C 0.000} C_DIS
LIN {X 49.203,Y -45.598,Z -152.739,A -90.000,B 90.000,C 0.000} C_DIS
LIN {X 49.555,Y -45.666,Z -152.678,A -90.000,B 90.000,C 0.000} C_DIS
LIN {X 50.347,Y -45.822,Z -152.562,A -90.000,B 90.000,C 0.000} C_DIS
LIN {X 50.981,Y -45.949,Z -152.495,A -90.000,B 90.000,C 0.000} C_DIS
LIN {X 51.382,Y -46.030,Z -152.465,A -90.000,B 90.000,C 0.000} C_DIS
LIN {X 51.587,Y -46.073,Z -152.453,A -90.000,B 90.000,C 0.000} C_DIS
LIN {X 51.674,Y -46.087,Z -152.450,A -90.000,B 90.000,C 0.000} C_DIS
LIN {X 52.175,Y -46.158,Z -152.439,A -90.000,B 90.000,C 0.000} C_DIS
LIN {X 52.656,Y -46.228,Z -152.444,A -90.000,B 90.000,C 0.000} C_DIS
LIN {X 53.238,Y -46.314,Z -152.465,A -90.000,B 90.000,C 0.000} C_DIS
LIN {X 53.572,Y -46.363,Z -152.487,A -90.000,B 90.000,C 0.000} C_DIS
LIN {X 54.105,Y -46.442,Z -152.534,A -90.000,B 90.000,C 0.000} C_DIS
LIN {X 54.494,Y -46.501,Z -152.578,A -90.000,B 90.000,C 0.000} C_DIS
LIN {X 54.602,Y -46.517,Z -152.593,A -90.000,B 90.000,C 0.000} C_DIS
LIN {X 55.191,Y -46.559,Z -152.684,A -90.000,B 90.000,C 0.000} C_DIS
LIN {X 55.490,Y -46.581,Z -152.739,A -90.000,B 90.000,C 0.000} C_DIS
LIN {X 55.822,Y -46.609,Z -152.804,A -90.000,B 90.000,C 0.000} C_DIS
LIN {X 56.327,Y -46.653,Z -152.919,A -90.000,B 90.000,C 0.000} C_DIS
LIN {X 56.839,Y -46.699,Z -153.051,A -90.000,B 90.000,C 0.000} C_DIS
LIN {X 57.154,Y -46.727,Z -153.137,A -90.000,B 90.000,C 0.000} C_DIS
LIN {X 57.355,Y -46.739,Z -153.198,A -90.000,B 90.000,C 0.000} C_DIS
LIN {X 57.489,Y -46.746,Z -153.239,A -90.000,B 90.000,C 0.000} C_DIS
LIN {X 57.589,Y -46.750,Z -153.271,A -90.000,B 90.000,C 0.000} C_DIS
LIN {X 58.150,Y -46.752,Z -153.462,A -90.000,B 90.000,C 0.000} C_DIS
LIN {X 58.686,Y -46.756,Z -153.665,A -90.000,B 90.000,C 0.000} C_DIS
LIN {X 59.247,Y -46.764,Z -153.896,A -90.000,B 90.000,C 0.000} C_DIS
LIN {X 59.510,Y -46.769,Z -154.013,A -90.000,B 90.000,C 0.000} C_DIS
LIN {X 60.026,Y -46.779,Z -154.258,A -90.000,B 90.000,C 0.000} C_DIS
LIN {X 60.198,Y -46.782,Z -154.346,A -90.000,B 90.000,C 0.000} C_DIS
LIN {X 60.272,Y -46.781,Z -154.383,A -90.000,B 90.000,C 0.000} C_DIS
LIN {X 60.571,Y -46.764,Z -154.539,A -90.000,B 90.000,C 0.000} C_DIS
LIN {X 61.029,Y -46.734,Z -154.797,A -90.000,B 90.000,C 0.000} C_DIS
LIN {X 61.479,Y -46.705,Z -155.067,A -90.000,B 90.000,C 0.000} C_DIS
LIN {X 61.920,Y -46.676,Z -155.346,A -90.000,B 90.000,C 0.000} C_DIS
LIN {X 62.445,Y -46.644,Z -155.704,A -90.000,B 90.000,C 0.000} C_DIS
LIN {X 62.933,Y -46.614,Z -156.063,A -90.000,B 90.000,C 0.000} C_DIS
LIN {X 63.265,Y -46.595,Z -156.324,A -90.000,B 90.000,C 0.000} C_DIS
LIN {X 63.405,Y -46.577,Z -156.436,A -90.000,B 90.000,C 0.000} C_DIS
LIN {X 63.694,Y -46.536,Z -156.681,A -90.000,B 90.000,C 0.000} C_DIS
LIN {X 63.868,Y -46.509,Z -156.830,A -90.000,B 90.000,C 0.000} C_DIS
LIN {X 64.166,Y -46.462,Z -157.100,A -90.000,B 90.000,C 0.000} C_DIS
LIN {X 64.623,Y -46.389,Z -157.536,A -90.000,B 90.000,C 0.000} C_DIS
LIN {X 65.001,Y -46.329,Z -157.924,A -90.000,B 90.000,C 0.000} C_DIS
LIN {X 65.464,Y -46.255,Z -158.430,A -90.000,B 90.000,C 0.000} C_DIS
LIN {X 65.516,Y -46.246,Z -158.489,A -90.000,B 90.000,C 0.000} C_DIS
LIN {X 65.976,Y -46.171,Z -159.036,A -90.000,B 90.000,C 0.000} C_DIS
LIN {X 66.163,Y -46.130,Z -159.277,A -90.000,B 90.000,C 0.000} C_DIS
LIN {X 66.362,Y -46.085,Z -159.540,A -90.000,B 90.000,C 0.000} C_DIS
LIN {X 66.455,Y -46.062,Z -159.665,A -90.000,B 90.000,C 0.000} C_DIS
LIN {X 66.595,Y -46.026,Z -159.864,A -90.000,B 90.000,C 0.000} C_DIS
LIN {X 66.814,Y -45.971,Z -160.182,A -90.000,B 90.000,C 0.000} C_DIS
LIN {X 67.035,Y -45.914,Z -160.517,A -90.000,B 90.000,C 0.000} C_DIS
LIN {X 67.084,Y -45.901,Z -160.593,A -90.000,B 90.000,C 0.000} C_DIS
LIN {X 67.269,Y -45.853,Z -160.894,A -90.000,B 90.000,C 0.000} C_DIS
LIN {X 67.447,Y -45.807,Z -161.196,A -90.000,B 90.000,C 0.000} C_DIS
LIN {X 67.549,Y -45.776,Z -161.373,A -90.000,B 90.000,C 0.000} C_DIS
LIN {X 67.769,Y -45.707,Z -161.775,A -90.000,B 90.000,C 0.000} C_DIS
LIN {X 68.005,Y -45.631,Z -162.241,A -90.000,B 90.000,C 0.000} C_DIS
LIN {X 68.180,Y -45.574,Z -162.609,A -90.000,B 90.000,C 0.000} C_DIS
LIN {X 68.372,Y -45.510,Z -163.037,A -90.000,B 90.000,C 0.000} C_DIS
LIN {X 68.575,Y -45.440,Z -163.521,A -90.000,B 90.000,C 0.000} C_DIS
LIN {X 68.730,Y -45.384,Z -163.929,A -90.000,B 90.000,C 0.000} C_DIS
LIN {X 68.883,Y -45.308,Z -164.367,A -90.000,B 90.000,C 0.000} C_DIS
LIN {X 68.883,Y -60.000,Z -164.367,A -90.000,B 90.000,C 0.000} C_DIS
LIN {X 49.513,Y -60.000,Z -150.703,A -90.000,B 90.000,C 0.000} C_DIS
LIN {X 49.513,Y -45.308,Z -150.703,A -90.000,B 90.000,C 0.000} C_DIS
LIN {X 49.685,Y -45.346,Z -150.677,A -90.000,B 90.000,C 0.000} C_DIS
LIN {X 50.196,Y -45.446,Z -150.604,A -90.000,B 90.000,C 0.000} C_DIS
LIN {X 50.907,Y -45.588,Z -150.529,A -90.000,B 90.000,C 0.000} C_DIS
LIN {X 51.341,Y -45.677,Z -150.497,A -90.000,B 90.000,C 0.000} C_DIS
LIN {X 51.589,Y -45.729,Z -150.483,A -90.000,B 90.000,C 0.000} C_DIS
LIN {X 52.236,Y -45.867,Z -150.461,A -90.000,B 90.000,C 0.000} C_DIS
LIN {X 52.445,Y -45.913,Z -150.461,A -90.000,B 90.000,C 0.000} C_DIS
LIN {X 52.795,Y -45.967,Z -150.466,A -90.000,B 90.000,C 0.000} C_DIS
LIN {X 53.405,Y -46.058,Z -150.488,A -90.000,B 90.000,C 0.000} C_DIS
LIN {X 53.786,Y -46.116,Z -150.514,A -90.000,B 90.000,C 0.000} C_DIS
LIN {X 54.383,Y -46.209,Z -150.567,A -90.000,B 90.000,C 0.000} C_DIS
LIN {X 54.811,Y -46.278,Z -150.616,A -90.000,B 90.000,C 0.000} C_DIS
LIN {X 55.315,Y -46.350,Z -150.689,A -90.000,B 90.000,C 0.000} C_DIS
LIN {X 55.566,Y -46.372,Z -150.728,A -90.000,B 90.000,C 0.000} C_DIS
LIN {X 55.890,Y -46.399,Z -150.788,A -90.000,B 90.000,C 0.000} C_DIS
LIN {X 56.277,Y -46.433,Z -150.865,A -90.000,B 90.000,C 0.000} C_DIS
LIN {X 56.840,Y -46.484,Z -150.993,A -90.000,B 90.000,C 0.000} C_DIS
LIN {X 57.380,Y -46.535,Z -151.133,A -90.000,B 90.000,C 0.000} C_DIS
LIN {X 57.777,Y -46.577,Z -151.242,A -90.000,B 90.000,C 0.000} C_DIS
LIN {X 57.889,Y -46.588,Z -151.276,A -90.000,B 90.000,C 0.000} C_DIS
LIN {X 58.074,Y -46.597,Z -151.332,A -90.000,B 90.000,C 0.000} C_DIS
LIN {X 58.370,Y -46.604,Z -151.430,A -90.000,B 90.000,C 0.000} C_DIS
LIN {X 58.855,Y -46.612,Z -151.596,A -90.000,B 90.000,C 0.000} C_DIS
